KUKA KRL program: MyProgram_205().src

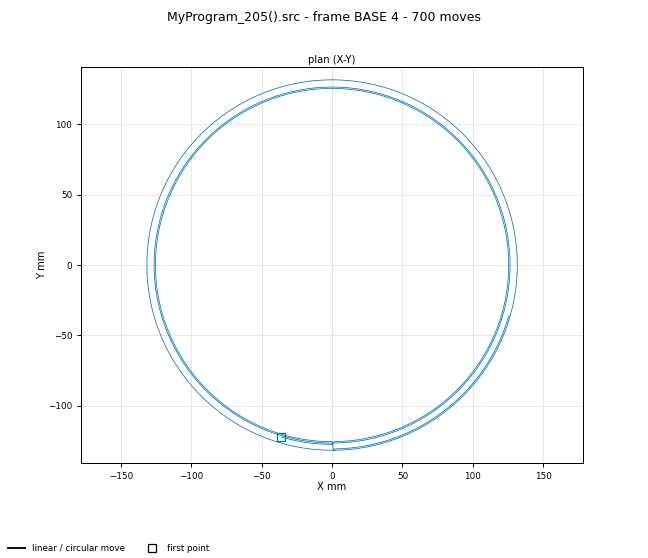
[picture p0: tool path of MyProgram_205().src in frame BASE 4, 700 of 700 moves have a stored position in this frame; points joined in program order, loops and branches not executed]
&ACCESS RVP
&REL 1
&PARAM TEMPLATE = C:\KRC\Roboter\Template\vorgabe
&PARAM EDITMASK = *
DEF MyProgram_205()
; ---- Setting reference (Base) ----
$BASE = BASE_DATA[4]

; --------------------------
; ---- Setting tool (TCP) ----
$TOOL = TOOL_DATA[3]
; --------------------------

$VEL.CP = VEL_APROX_PRINT
Startdeposition()
$VEL.CP = VEL_PRINT
LIN {X -36.0341,Y -122.2263,Z 146,A -108.5004,B 22.4031,C -0.9389,E1 22.3779,E2 195.6452} C_DIS
LIN {X -32.6607,Y -123.1706,Z 146,A -106.9156,B 22.4031,C -0.9383,E1 22.3822,E2 194.0592} C_DIS
LIN {X -28.9305,Y -124.1009,Z 146,A -105.1124,B 22.4031,C -0.9406,E1 22.3871,E2 192.2472} C_DIS
LIN {X -25.3241,Y -124.8856,Z 146,A -103.5291,B 22.4031,C -0.9365,E1 22.3914,E2 190.6725} C_DIS
LIN {X -21.3618,Y -125.6246,Z 146,A -101.0453,B 22.402,C -0.9659,E1 22.3984,E2 188.1089} C_DIS
LIN {X -16.3761,Y -126.3708,Z 146,A -99.4873,B 22.4033,C -0.9336,E1 22.4025,E2 186.6342} C_DIS
LIN {X -12.7363,Y -126.7906,Z 146,A -97.3876,B 22.4025,C -0.9536,E1 22.4085,E2 184.4806} C_DIS
LIN {X -9.0386,Y -127.1067,Z 146,A -96.2108,B 22.4034,C -0.9316,E1 22.4116,E2 183.3613} C_DIS
LIN {X -2.4319,Y -127.4047,Z 146,A -93.38,B 22.4036,C -0.9253,E1 22.4195,E2 180.5461} C_DIS
LIN {X 0.9115,Y -127.3964,Z 146,A -91.8987,B 22.4036,C -0.925,E1 22.4237,E2 179.0657} C_DIS
Enddeposition()
LIN {X 0.9115,Y -127.3964,Z 146,A -91.8987,B 22.4036,C -0.925,E1 22.4237,E2 179.0657} C_DIS
Startdeposition()
$VEL.CP = VEL_PRINT
LIN {X -0.2002,Y -126.4714,Z 146,A -92.567,B 21.3921,C -0.7578,E1 21.404,E2 180.0625} C_DIS
LIN {X -3.5171,Y -126.4217,Z 146,A -94.2559,B 21.3924,C -0.7499,E1 21.3992,E2 181.7734} C_DIS
LIN {X -7.0125,Y -126.2777,Z 146,A -95.5952,B 21.3921,C -0.76,E1 21.3955,E2 183.0853} C_DIS
LIN {X -11.0098,Y -125.9909,Z 146,A -97.3605,B 21.392,C -0.7622,E1 21.3906,E2 184.8454} C_DIS
LIN {X -14.3334,Y -125.6573,Z 146,A -99.0886,B 21.3923,C -0.7535,E1 21.3858,E2 186.5988} C_DIS
LIN {X -19.2644,Y -124.9946,Z 146,A -101.275,B 21.3922,C -0.7568,E1 21.3797,E2 188.778} C_DIS
LIN {X -22.4995,Y -124.4531,Z 146,A -102.727,B 21.3922,C -0.7588,E1 21.3758,E2 190.2264} C_DIS
LIN {X -26.5997,Y -123.6414,Z 146,A -104.6613,B 21.3922,C -0.7579,E1 21.3705,E2 192.1657} C_DIS
LIN {X -29.8792,Y -122.8903,Z 146,A -106.087,B 21.392,C -0.7628,E1 21.3666,E2 193.5803} C_DIS
LIN {X -32.8395,Y -122.1326,Z 146,A -107.6058,B 21.3921,C -0.7581,E1 21.3625,E2 195.1146} C_DIS
LIN {X -37.1654,Y -120.8862,Z 146,A -109.654,B 21.3921,C -0.7592,E1 21.357,E2 197.1639} C_DIS
LIN {X -42.6541,Y -119.0604,Z 146,A -111.9494,B 21.3916,C -0.7746,E1 21.351,E2 199.4219} C_DIS
LIN {X -48.2784,Y -116.8936,Z 146,A -114.7855,B 21.3916,C -0.7729,E1 21.3436,E2 202.27} C_DIS
LIN {X -50.5646,Y -115.9227,Z 146,A -115.9953,B 21.3917,C -0.7707,E1 21.3405,E2 203.4892} C_DIS
LIN {X -53.5348,Y -114.5816,Z 146,A -117.5184,B 21.3917,C -0.7705,E1 21.3366,E2 205.0174} C_DIS
LIN {X -56.4308,Y -113.1836,Z 146,A -118.9521,B 21.3917,C -0.7732,E1 21.333,E2 206.448} C_DIS
LIN {X -59.1321,Y -111.7954,Z 146,A -120.3858,B 21.3917,C -0.7727,E1 21.3294,E2 207.8879} C_DIS
LIN {X -62.7954,Y -109.7812,Z 146,A -122.3752,B 21.3917,C -0.7714,E1 21.3246,E2 209.8876} C_DIS
LIN {X -66.3971,Y -107.6414,Z 146,A -124.2637,B 21.3916,C -0.7746,E1 21.3201,E2 211.7743} C_DIS
LIN {X -69.8004,Y -105.4664,Z 146,A -126.1081,B 21.3915,C -0.7769,E1 21.3157,E2 213.6195} C_DIS
LIN {X -77.0801,Y -100.2691,Z 146,A -129.8585,B 21.3908,C -0.7957,E1 21.3074,E2 217.3336} C_DIS
LIN {X -79.9121,Y -98.0267,Z 146,A -131.4603,B 21.3907,C -0.8001,E1 21.3038,E2 218.9304} C_DIS
LIN {X -83.4451,Y -95.0379,Z 146,A -133.9643,B 21.3911,C -0.788,E1 21.2984,E2 221.4794} C_DIS
LIN {X -86.6555,Y -92.1196,Z 146,A -135.9206,B 21.391,C -0.7923,E1 21.2944,E2 223.4332} C_DIS
LIN {X -89.7097,Y -89.1478,Z 146,A -137.8436,B 21.3908,C -0.7966,E1 21.2906,E2 225.3539} C_DIS
LIN {X -92.795,Y -85.9323,Z 146,A -139.8605,B 21.3906,C -0.8011,E1 21.2867,E2 227.3689} C_DIS
LIN {X -95.6026,Y -82.7974,Z 146,A -141.8312,B 21.3906,C -0.8029,E1 21.2831,E2 229.3453} C_DIS
LIN {X -98.4968,Y -79.3318,Z 146,A -144.1879,B 21.3908,C -0.7956,E1 21.2789,E2 231.7351} C_DIS
LIN {X -100.8297,Y -76.3451,Z 146,A -145.3981,B 21.39,C -0.8194,E1 21.2769,E2 232.8867} C_DIS
LIN {X -103.3227,Y -72.9355,Z 146,A -147.5852,B 21.3902,C -0.8135,E1 21.2733,E2 235.1026} C_DIS
LIN {X -105.7732,Y -69.3344,Z 146,A -149.5373,B 21.39,C -0.8193,E1 21.2703,E2 237.0503} C_DIS
LIN {X -108.0776,Y -65.6847,Z 146,A -151.4874,B 21.3898,C -0.8246,E1 21.2674,E2 238.9977} C_DIS
LIN {X -112.2795,Y -58.2101,Z 146,A -155.097,B 21.389,C -0.8456,E1 21.2626,E2 242.5719} C_DIS
LIN {X -113.9687,Y -54.8262,Z 146,A -156.7959,B 21.3888,C -0.8509,E1 21.2605,E2 244.2672} C_DIS
LIN {X -115.4791,Y -51.568,Z 146,A -158.6195,B 21.3889,C -0.8479,E1 21.2583,E2 246.1109} C_DIS
LIN {X -116.6221,Y -48.9286,Z 146,A -159.9466,B 21.3889,C -0.8507,E1 21.2569,E2 247.4391} C_DIS
LIN {X -117.8749,Y -45.8278,Z 146,A -161.5498,B 21.3888,C -0.8516,E1 21.2552,E2 249.0502} C_DIS
LIN {X -119.1113,Y -42.513,Z 146,A -163.0181,B 21.3884,C -0.8615,E1 21.2538,E2 250.5014} C_DIS
LIN {X -119.9494,Y -40.0857,Z 146,A -164.511,B 21.3888,C -0.8523,E1 21.2525,E2 252.0296} C_DIS
LIN {X -121.4192,Y -35.3851,Z 146,A -166.5476,B 21.3882,C -0.8664,E1 21.2509,E2 254.0414} C_DIS
LIN {X -122.6901,Y -30.6928,Z 146,A -168.844,B 21.3881,C -0.8694,E1 21.2492,E2 256.3453} C_DIS
LIN {X -123.6495,Y -26.5625,Z 146,A -170.6967,B 21.3878,C -0.8779,E1 21.2481,E2 258.1875} C_DIS
LIN {X -124.2918,Y -23.3759,Z 146,A -172.1355,B 21.3875,C -0.8837,E1 21.2473,E2 259.6204} C_DIS
LIN {X -124.9553,Y -19.5185,Z 146,A -173.9521,B 21.3874,C -0.8876,E1 21.2465,E2 261.4393} C_DIS
LIN {X -125.4853,Y -15.7689,Z 146,A -175.8504,B 21.3874,C -0.886,E1 21.2458,E2 263.3554} C_DIS
LIN {X -125.9635,Y -11.3339,Z 146,A -177.6417,B 21.3868,C -0.901,E1 21.2453,E2 265.118} C_DIS
LIN {X -126.1813,Y -8.5712,Z 146,A -179.0869,B 21.387,C -0.8978,E1 21.245,E2 266.5824} C_DIS
LIN {X -126.3845,Y -4.6711,Z 146,A 179.1289,B 21.3868,C -0.9028,E1 21.2448,E2 268.3655} C_DIS
LIN {X -126.4753,Y -0.0344,Z 146,A 177.1063,B 21.3864,C -0.9124,E1 21.2448,E2 270.3762} C_DIS
LIN {X -126.381,Y 4.7613,Z 146,A 174.9068,B 21.3861,C -0.9184,E1 21.2448,E2 272.5751} C_DIS
LIN {X -126.164,Y 8.8087,Z 146,A 173.0434,B 21.3859,C -0.9232,E1 21.2452,E2 274.4385} C_DIS
LIN {X -125.8611,Y 12.4043,Z 146,A 171.377,B 21.3858,C -0.9272,E1 21.2456,E2 276.1058} C_DIS
LIN {X -125.3982,Y 16.4334,Z 146,A 169.5121,B 21.3856,C -0.932,E1 21.2463,E2 277.9708} C_DIS
LIN {X -124.7679,Y 20.6819,Z 146,A 167.6246,B 21.3852,C -0.9403,E1 21.2471,E2 279.8486} C_DIS
LIN {X -124.1633,Y 24.048,Z 146,A 165.628,B 21.3857,C -0.9283,E1 21.2481,E2 281.8923} C_DIS
LIN {X -123.3778,Y 27.7993,Z 146,A 164.5101,B 21.3845,C -0.9571,E1 21.2488,E2 282.9386} C_DIS
LIN {X -122.4488,Y 31.6436,Z 146,A 162.5398,B 21.3845,C -0.9559,E1 21.2501,E2 284.9259} C_DIS
LIN {X -121.5509,Y 34.9355,Z 146,A 160.7569,B 21.3848,C -0.9517,E1 21.2514,E2 286.7326} C_DIS
LIN {X -120.1897,Y 39.3641,Z 146,A 158.9282,B 21.384,C -0.9684,E1 21.253,E2 288.5278} C_DIS
LIN {X -119.2918,Y 42.0064,Z 146,A 157.443,B 21.3842,C -0.9639,E1 21.2543,E2 290.0354} C_DIS
LIN {X -117.8314,Y 45.9397,Z 146,A 155.6344,B 21.3838,C -0.9732,E1 21.2561,E2 291.8306} C_DIS
LIN {X -116.6725,Y 48.808,Z 146,A 153.266,B 21.3852,C -0.941,E1 21.2588,E2 294.3034} C_DIS
LIN {X -114.0463,Y 54.6639,Z 146,A 151.2733,B 21.3834,C -0.9839,E1 21.261,E2 296.1905} C_DIS
LIN {X -111.7773,Y 59.1664,Z 146,A 149.0935,B 21.3829,C -0.9945,E1 21.2638,E2 298.355} C_DIS
LIN {X -110.0652,Y 62.2974,Z 146,A 147.3565,B 21.3829,C -0.9945,E1 21.2662,E2 300.1029} C_DIS
LIN {X -108.057,Y 65.7187,Z 146,A 145.4612,B 21.3829,C -0.9959,E1 21.2689,E2 302.0062} C_DIS
LIN {X -105.7694,Y 69.34,Z 146,A 143.5175,B 21.3826,C -1.0011,E1 21.2718,E2 303.9471} C_DIS
LIN {X -103.2904,Y 72.9812,Z 146,A 141.6623,B 21.3821,C -1.0118,E1 21.2747,E2 305.7835} C_DIS
LIN {X -101.3754,Y 75.6186,Z 146,A 140.0515,B 21.3821,C -1.0106,E1 21.2774,E2 307.407} C_DIS
LIN {X -98.7229,Y 79.051,Z 146,A 138.2823,B 21.3816,C -1.0232,E1 21.2804,E2 309.1514} C_DIS
LIN {X -96.8688,Y 81.3116,Z 146,A 136.7318,B 21.3818,C -1.018,E1 21.2832,E2 310.7249} C_DIS
LIN {X -94.0244,Y 84.5851,Z 146,A 134.6597,B 21.3818,C -1.0187,E1 21.2871,E2 312.806} C_DIS
LIN {X -90.6963,Y 88.1441,Z 146,A 132.5897,B 21.3813,C -1.0293,E1 21.291,E2 314.8575} C_DIS
LIN {X -87.9405,Y 90.8935,Z 146,A 130.7775,B 21.3813,C -1.0316,E1 21.2946,E2 316.6725} C_DIS
LIN {X -85.0052,Y 93.6444,Z 146,A 128.8415,B 21.3813,C -1.0314,E1 21.2986,E2 318.6184} C_DIS
LIN {X -81.8441,Y 96.4194,Z 146,A 127.0047,B 21.3809,C -1.0382,E1 21.3025,E2 320.4449} C_DIS
LIN {X -78.8892,Y 98.8518,Z 146,A 125.3343,B 21.3806,C -1.0443,E1 21.3061,E2 322.1059} C_DIS
LIN {X -75.836,Y 101.2136,Z 146,A 123.5138,B 21.3806,C -1.0451,E1 21.3101,E2 323.932} C_DIS
LIN {X -71.8456,Y 104.084,Z 146,A 121.2314,B 21.3805,C -1.0473,E1 21.3154,E2 326.2177} C_DIS
LIN {X -68.6655,Y 106.2086,Z 146,A 119.5061,B 21.3803,C -1.0509,E1 21.3194,E2 327.94} C_DIS
LIN {X -65.3364,Y 108.2881,Z 146,A 117.7441,B 21.3801,C -1.0547,E1 21.3236,E2 329.698} C_DIS
LIN {X -62.0308,Y 110.215,Z 146,A 116.0512,B 21.3799,C -1.0593,E1 21.3277,E2 331.3842} C_DIS
LIN {X -58.7576,Y 111.992,Z 146,A 114.4151,B 21.3797,C -1.0641,E1 21.3317,E2 333.0126} C_DIS
LIN {X -55.9636,Y 113.414,Z 146,A 112.9155,B 21.3797,C -1.0632,E1 21.3354,E2 334.5194} C_DIS
LIN {X -52.2563,Y 115.1712,Z 146,A 111.1648,B 21.3794,C -1.0702,E1 21.3398,E2 336.256} C_DIS
LIN {X -49.3423,Y 116.4493,Z 146,A 109.7278,B 21.3794,C -1.0724,E1 21.3435,E2 337.691} C_DIS
LIN {X -46.2318,Y 117.7179,Z 146,A 107.792,B 21.38,C -1.0581,E1 21.3486,E2 339.6712} C_DIS
LIN {X -43.1661,Y 118.8758,Z 146,A 106.861,B 21.3789,C -1.0818,E1 21.3509,E2 340.5391} C_DIS
LIN {X -38.6181,Y 120.4299,Z 146,A 104.0568,B 21.3799,C -1.0595,E1 21.3585,E2 343.4109} C_DIS
LIN {X -35.1143,Y 121.4985,Z 146,A 102.8457,B 21.379,C -1.079,E1 21.3616,E2 344.5707} C_DIS
LIN {X -32.1662,Y 122.3121,Z 146,A 101.4603,B 21.379,C -1.0804,E1 21.3654,E2 345.9548} C_DIS
LIN {X -29.4254,Y 122.9997,Z 146,A 100.0934,B 21.379,C -1.0781,E1 21.3691,E2 347.3303} C_DIS
LIN {X -26.4415,Y 123.6756,Z 146,A 98.758,B 21.3789,C -1.0813,E1 21.3727,E2 348.6589} C_DIS
LIN {X -23.5848,Y 124.2519,Z 146,A 97.3859,B 21.3789,C -1.0802,E1 21.3765,E2 350.0358} C_DIS
LIN {X -19.2825,Y 124.9918,Z 146,A 95.384,B 21.3789,C -1.0806,E1 21.382,E2 352.0388} C_DIS
LIN {X -14.8809,Y 125.592,Z 146,A 93.3443,B 21.3789,C -1.0806,E1 21.3877,E2 354.0802} C_DIS
LIN {X -11.5392,Y 125.9442,Z 146,A 91.8914,B 21.3787,C -1.0841,E1 21.3917,E2 355.5245} C_DIS
LIN {X -7.5118,Y 126.2475,Z 146,A 90.1618,B 21.3785,C -1.0889,E1 21.3965,E2 357.2417} C_DIS
LIN {X -4.6049,Y 126.3871,Z 146,A 88.8159,B 21.3785,C -1.0882,E1 21.4002,E2 358.5899} C_DIS
LIN {X -1.3758,Y 126.4649,Z 146,A 87.2194,B 21.3788,C -1.083,E1 21.4047,E2 360.2007} C_DIS
LIN {X 2.7721,Y 126.4415,Z 146,A 85.4789,B 21.3785,C -1.0889,E1 21.4095,E2 361.9247} C_DIS
LIN {X 7.4851,Y 126.2492,Z 146,A 83.1677,B 21.3789,C -1.0818,E1 21.416,E2 364.2545} C_DIS
LIN {X 11.0113,Y 125.9908,Z 146,A 81.7032,B 21.3786,C -1.0873,E1 21.4201,E2 365.703} C_DIS
LIN {X 14.5679,Y 125.6293,Z 146,A 79.9193,B 21.3789,C -1.0802,E1 21.4251,E2 367.5049} C_DIS
LIN {X 18.102,Y 125.1684,Z 146,A 78.4196,B 21.3787,C -1.0845,E1 21.4292,E2 368.9912} C_DIS
LIN {X 22.1034,Y 124.524,Z 146,A 76.484,B 21.379,C -1.0798,E1 21.4345,E2 370.9376} C_DIS
LIN {X 25.5845,Y 123.856,Z 146,A 75.0215,B 21.3787,C -1.085,E1 21.4385,E2 372.3837} C_DIS
LIN {X 28.2648,Y 123.2714,Z 146,A 73.7554,B 21.3787,C -1.0833,E1 21.4419,E2 373.6523} C_DIS
LIN {X 31.3296,Y 122.5285,Z 146,A 72.3059,B 21.3789,C -1.0816,E1 21.4459,E2 375.1039} C_DIS
LIN {X 35.1324,Y 121.4932,Z 146,A 70.4772,B 21.379,C -1.0785,E1 21.4508,E2 376.9375} C_DIS
LIN {X 39.9482,Y 119.9952,Z 146,A 68.5858,B 21.3783,C -1.0932,E1 21.4557,E2 378.7844} C_DIS
LIN {X 45.5483,Y 117.9836,Z 146,A 65.7798,B 21.3787,C -1.0861,E1 21.4632,E2 381.6031} C_DIS
LIN {X 48.8944,Y 116.6364,Z 146,A 63.9332,B 21.3792,C -1.0754,E1 21.468,E2 383.474} C_DIS
LIN {X 52.184,Y 115.2036,Z 146,A 62.3271,B 21.3792,C -1.0743,E1 21.4721,E2 385.0783} C_DIS
LIN {X 54.7767,Y 113.9924,Z 146,A 61.0283,B 21.3792,C -1.0727,E1 21.4753,E2 386.3776} C_DIS
LIN {X 58.1819,Y 112.2943,Z 146,A 59.1911,B 21.3796,C -1.0656,E1 21.48,E2 388.2281} C_DIS
LIN {X 62.1945,Y 110.123,Z 146,A 57.2128,B 21.3796,C -1.0665,E1 21.4848,E2 390.1971} C_DIS
LIN {X 65.5406,Y 108.1647,Z 146,A 55.509,B 21.3796,C -1.0661,E1 21.4888,E2 391.8956} C_DIS
LIN {X 68.6592,Y 106.2127,Z 146,A 53.774,B 21.3799,C -1.0606,E1 21.493,E2 393.639} C_DIS
LIN {X 71.951,Y 104.0112,Z 146,A 51.9083,B 21.3802,C -1.0546,E1 21.4973,E2 395.5138} C_DIS
LIN {X 75.3343,Y 101.5872,Z 146,A 50.0448,B 21.3802,C -1.0522,E1 21.5015,E2 397.3757} C_DIS
LIN {X 78.1149,Y 99.4646,Z 146,A 48.5612,B 21.3802,C -1.0537,E1 21.5047,E2 398.8488} C_DIS
LIN {X 80.9804,Y 97.1467,Z 146,A 46.7924,B 21.3805,C -1.0463,E1 21.5086,E2 400.6299} C_DIS
LIN {X 84.3041,Y 94.2761,Z 146,A 44.8386,B 21.3807,C -1.0439,E1 21.5127,E2 402.581} C_DIS
LIN {X 87.2293,Y 91.5764,Z 146,A 43.0399,B 21.3808,C -1.0404,E1 21.5163,E2 404.3804} C_DIS
LIN {X 90.1747,Y 88.6775,Z 146,A 41.2654,B 21.3808,C -1.0407,E1 21.5198,E2 406.1452} C_DIS
LIN {X 92.9177,Y 85.7994,Z 146,A 39.5495,B 21.3808,C -1.0404,E1 21.5231,E2 407.853} C_DIS
LIN {X 95.3156,Y 83.127,Z 146,A 37.7882,B 21.3813,C -1.0309,E1 21.5264,E2 409.6309} C_DIS
LIN {X 98.1919,Y 79.7099,Z 146,A 35.7281,B 21.3815,C -1.0245,E1 21.5301,E2 411.697} C_DIS
LIN {X 100.9079,Y 76.2415,Z 146,A 33.8091,B 21.3816,C -1.0231,E1 21.5333,E2 413.6092} C_DIS
LIN {X 103.467,Y 72.7309,Z 146,A 31.953,B 21.3816,C -1.0231,E1 21.5363,E2 415.4545} C_DIS
LIN {X 105.205,Y 70.193,Z 146,A 30.5018,B 21.3819,C -1.0171,E1 21.5386,E2 416.9137} C_DIS
LIN {X 107.5118,Y 66.6065,Z 146,A 28.6131,B 21.382,C -1.0139,E1 21.5414,E2 418.7996} C_DIS
LIN {X 109.4763,Y 63.3254,Z 146,A 26.7412,B 21.3825,C -1.0032,E1 21.5441,E2 420.6892} C_DIS
LIN {X 111.3301,Y 60.0067,Z 146,A 25.0158,B 21.3827,C -0.9984,E1 21.5464,E2 422.417} C_DIS
LIN {X 113.4712,Y 55.8477,Z 146,A 23.0715,B 21.3827,C -1.0003,E1 21.5488,E2 424.3438} C_DIS
LIN {X 114.9056,Y 52.8341,Z 146,A 21.6136,B 21.3827,C -0.9985,E1 21.5506,E2 425.7974} C_DIS
LIN {X 117.6429,Y 46.4246,Z 146,A 18.5231,B 21.383,C -0.9924,E1 21.5539,E2 428.8843} C_DIS
LIN {X 118.6502,Y 43.7857,Z 146,A 17.204,B 21.3832,C -0.9869,E1 21.5552,E2 430.2096} C_DIS
LIN {X 119.597,Y 41.1262,Z 146,A 15.6046,B 21.384,C -0.9689,E1 21.5567,E2 431.8474} C_DIS
LIN {X 121.2732,Y 35.884,Z 146,A 13.3951,B 21.3838,C -0.9741,E1 21.5585,E2 434.0279} C_DIS
LIN {X 122.1777,Y 32.6703,Z 146,A 11.93,B 21.3839,C -0.9716,E1 21.5596,E2 435.4896} C_DIS
LIN {X 122.9913,Y 29.4602,Z 146,A 10.424,B 21.3841,C -0.9668,E1 21.5606,E2 436.9984} C_DIS
LIN {X 123.696,Y 26.347,Z 146,A 9.0665,B 21.3841,C -0.9663,E1 21.5614,E2 438.3478} C_DIS
LIN {X 124.2447,Y 23.6226,Z 146,A 7.7618,B 21.3844,C -0.9604,E1 21.5621,E2 439.6596} C_DIS
LIN {X 124.8827,Y 19.9873,Z 146,A 6.1731,B 21.3844,C -0.9589,E1 21.5628,E2 441.2413} C_DIS
LIN {X 125.3847,Y 16.5368,Z 146,A 4.5913,B 21.3847,C -0.9539,E1 21.5635,E2 442.8256} C_DIS
LIN {X 125.8017,Y 13,Z 146,A 2.9894,B 21.3849,C -0.9494,E1 21.564,E2 444.4287} C_DIS
LIN {X 126.0952,Y 9.751,Z 146,A 1.5779,B 21.3849,C -0.9477,E1 21.5643,E2 445.8348} C_DIS
LIN {X 126.2638,Y 7.2469,Z 146,A 0.1224,B 21.3857,C -0.9298,E1 21.5645,E2 447.3287} C_DIS
LIN {X 126.4447,Y 2.6084,Z 146,A -1.8242,B 21.3857,C -0.9301,E1 21.5647,E2 449.2606} C_DIS
LIN {X 126.4634,Y -1.4399,Z 146,A -3.6754,B 21.3859,C -0.9235,E1 21.5647,E2 451.1168} C_DIS
LIN {X 126.3687,Y -5.0768,Z 146,A -5.2969,B 21.3861,C -0.9195,E1 21.5645,E2 452.7378} C_DIS
LIN {X 126.1804,Y -8.5843,Z 146,A -6.8164,B 21.3861,C -0.9176,E1 21.5643,E2 454.2516} C_DIS
LIN {X 125.9003,Y -11.996,Z 146,A -8.3839,B 21.3864,C -0.912,E1 21.5639,E2 455.8235} C_DIS
LIN {X 125.3751,Y -16.6097,Z 146,A -10.2401,B 21.3862,C -0.9164,E1 21.5633,E2 457.6546} C_DIS
LIN {X 124.9979,Y -19.2433,Z 146,A -11.6731,B 21.3868,C -0.9023,E1 21.5627,E2 459.1159} C_DIS
LIN {X 124.3558,Y -23.0412,Z 146,A -13.296,B 21.3868,C -0.9023,E1 21.5619,E2 460.7276} C_DIS
LIN {X 123.5962,Y -26.8094,Z 146,A -15.1438,B 21.3872,C -0.892,E1 21.5608,E2 462.5906} C_DIS
LIN {X 122.793,Y -30.2827,Z 146,A -16.6457,B 21.3872,C -0.892,E1 21.5599,E2 464.0822} C_DIS
LIN {X 121.8501,Y -33.8719,Z 146,A -18.8983,B 21.3884,C -0.8613,E1 21.5582,E2 466.4032} C_DIS
LIN {X 120.5843,Y -38.135,Z 146,A -20.1527,B 21.3873,C -0.889,E1 21.5572,E2 467.5734} C_DIS
LIN {X 119.7154,Y -40.7847,Z 146,A -21.5355,B 21.3877,C -0.8797,E1 21.556,E2 468.9723} C_DIS
LIN {X 118.3362,Y -44.6241,Z 146,A -23.4349,B 21.388,C -0.8718,E1 21.5541,E2 470.8806} C_DIS
LIN {X 116.8715,Y -48.3314,Z 146,A -25.6354,B 21.3889,C -0.8487,E1 21.5518,E2 473.1295} C_DIS
LIN {X 115.422,Y -51.6956,Z 146,A -26.9406,B 21.3885,C -0.8596,E1 21.5503,E2 474.3967} C_DIS
LIN {X 113.7971,Y -55.1856,Z 146,A -28.5736,B 21.3885,C -0.8594,E1 21.5484,E2 476.0198} C_DIS
LIN {X 112.5392,Y -57.7039,Z 146,A -29.9715,B 21.3888,C -0.8502,E1 21.5466,E2 477.4339} C_DIS
LIN {X 110.82,Y -60.9443,Z 146,A -31.6223,B 21.389,C -0.8459,E1 21.5444,E2 479.0863} C_DIS
LIN {X 109.0869,Y -63.9939,Z 146,A -33.1803,B 21.3891,C -0.8427,E1 21.5422,E2 480.6432} C_DIS
LIN {X 106.8228,Y -67.7059,Z 146,A -35.435,B 21.3898,C -0.8246,E1 21.5388,E2 482.9339} C_DIS
LIN {X 104.8688,Y -70.6948,Z 146,A -36.6955,B 21.3894,C -0.836,E1 21.5369,E2 484.1559} C_DIS
LIN {X 103.3679,Y -72.8713,Z 146,A -37.9082,B 21.3895,C -0.832,E1 21.535,E2 485.3722} C_DIS
LIN {X 100.9849,Y -76.1393,Z 146,A -39.9844,B 21.3901,C -0.8163,E1 21.5315,E2 487.4794} C_DIS
LIN {X 99.006,Y -78.6955,Z 146,A -41.1237,B 21.3897,C -0.8269,E1 21.5296,E2 488.5834} C_DIS
LIN {X 94.5241,Y -84.0266,Z 146,A -44.3113,B 21.39,C -0.8174,E1 21.5238,E2 491.7797} C_DIS
LIN {X 89.5198,Y -89.3389,Z 146,A -48.2395,B 21.3913,C -0.7821,E1 21.516,E2 495.7843} C_DIS
LIN {X 85.8463,Y -92.8744,Z 146,A -49.9498,B 21.3906,C -0.803,E1 21.5127,E2 497.4291} C_DIS
LIN {X 80.2118,Y -97.7817,Z 146,A -53.6721,B 21.3914,C -0.7807,E1 21.5046,E2 501.1951} C_DIS
LIN {X 77.1053,Y -100.2499,Z 146,A -55.1228,B 21.391,C -0.7921,E1 21.5015,E2 502.6084} C_DIS
LIN {X 72.465,Y -103.6536,Z 146,A -57.5038,B 21.3908,C -0.7967,E1 21.4962,E2 504.9667} C_DIS
LIN {X 70.5141,Y -104.9907,Z 146,A -58.7664,B 21.3912,C -0.7863,E1 21.4932,E2 506.2528} C_DIS
LIN {X 66.9866,Y -107.2753,Z 146,A -60.6679,B 21.3912,C -0.7828,E1 21.4887,E2 508.1564} C_DIS
LIN {X 63.1023,Y -109.6054,Z 146,A -62.7171,B 21.3914,C -0.7793,E1 21.4838,E2 510.2079} C_DIS
LIN {X 59.0055,Y -111.8619,Z 146,A -64.5512,B 21.3911,C -0.7881,E1 21.4794,E2 512.0115} C_DIS
LIN {X 56.6188,Y -113.0908,Z 146,A -66.0383,B 21.3916,C -0.7743,E1 21.4756,E2 513.5314} C_DIS
LIN {X 50.8017,Y -115.8202,Z 146,A -69.0261,B 21.3918,C -0.7666,E1 21.468,E2 516.5313} C_DIS
LIN {X 46.9994,Y -117.4131,Z 146,A -70.7002,B 21.3916,C -0.7724,E1 21.4637,E2 518.185} C_DIS
LIN {X 43.1653,Y -118.8761,Z 146,A -73.0884,B 21.3925,C -0.7473,E1 21.4573,E2 520.6359} C_DIS
LIN {X 38.9648,Y -120.3192,Z 146,A -74.4068,B 21.3916,C -0.7746,E1 21.454,E2 521.8766} C_DIS
LIN {X 35.1139,Y -121.4987,Z 146,A -76.4604,B 21.392,C -0.7628,E1 21.4484,E2 523.9584} C_DIS
LIN {X 31.224,Y -122.5553,Z 146,A -78.2182,B 21.392,C -0.7639,E1 21.4437,E2 525.7099} C_DIS
LIN {X 27.7361,Y -123.3922,Z 146,A -79.9259,B 21.3921,C -0.7588,E1 21.439,E2 527.4285} C_DIS
LIN {X 23.6769,Y -124.2343,Z 146,A -81.6893,B 21.392,C -0.7622,E1 21.4342,E2 529.1802} C_DIS
LIN {X 20.477,Y -124.8021,Z 146,A -83.2544,B 21.3922,C -0.7572,E1 21.4299,E2 530.757} C_DIS
LIN {X 16.4443,Y -125.3968,Z 146,A -84.764,B 21.3917,C -0.7703,E1 21.4258,E2 532.2292} C_DIS
LIN {X 13.6399,Y -125.7328,Z 146,A -86.2982,B 21.3921,C -0.7587,E1 21.4215,E2 533.7936} C_DIS
LIN {X 9.6443,Y -126.103,Z 146,A -88.2666,B 21.3924,C -0.7515,E1 21.4159,E2 535.7805} C_DIS
LIN {X 3.5217,Y -126.4215,Z 146,A -90.838,B 21.3921,C -0.7593,E1 21.4088,E2 538.3297} C_DIS
LIN {X 0.9047,Y -126.4634,Z 146,A -91.6983,B 21.3916,C -0.7727,E1 21.4065,E2 539.153} C_DIS
Enddeposition()
LIN {X 0.9047,Y -126.4634,Z 146,A -91.6983,B 21.3916,C -0.7727,E1 21.4065,E2 539.153} C_DIS
Startdeposition()
$VEL.CP = VEL_PRINT
LIN {X 1.5275,Y -125.5056,Z 146,A -90.6951,B 20.265,C -0.6363,E1 20.2782,E2 538.4061} C_DIS
LIN {X 4.5983,Y -125.4297,Z 146,A -89.3182,B 20.265,C -0.6358,E1 20.282,E2 537.0313} C_DIS
LIN {X 7.9101,Y -125.2642,Z 146,A -87.8871,B 20.265,C -0.633,E1 20.286,E2 535.6088} C_DIS
LIN {X 11.0165,Y -125.03,Z 146,A -86.458,B 20.265,C -0.6339,E1 20.29,E2 534.178} C_DIS
LIN {X 13.8261,Y -124.7503,Z 146,A -85.1681,B 20.265,C -0.6347,E1 20.2936,E2 532.8871} C_DIS
LIN {X 17.1185,Y -124.3423,Z 146,A -83.6966,B 20.265,C -0.6338,E1 20.2976,E2 531.4196} C_DIS
LIN {X 19.9422,Y -123.9212,Z 146,A -82.2521,B 20.2649,C -0.6404,E1 20.3016,E2 529.9579} C_DIS
LIN {X 22.9726,Y -123.3947,Z 146,A -80.86,B 20.2649,C -0.641,E1 20.3055,E2 528.566} C_DIS
LIN {X 26.2347,Y -122.7413,Z 146,A -79.4247,B 20.2649,C -0.6389,E1 20.3094,E2 527.1391} C_DIS
LIN {X 29.2363,Y -122.0609,Z 146,A -77.8981,B 20.2647,C -0.6451,E1 20.3136,E2 525.5972} C_DIS
LIN {X 33.477,Y -120.9669,Z 146,A -75.967,B 20.2647,C -0.6443,E1 20.3188,E2 523.6723} C_DIS
LIN {X 36.6722,Y -120.0364,Z 146,A -74.4493,B 20.2647,C -0.6459,E1 20.3228,E2 522.1534} C_DIS
LIN {X 40.6153,Y -118.7613,Z 146,A -72.5021,B 20.2645,C -0.6504,E1 20.328,E2 520.198} C_DIS
LIN {X 44.6291,Y -117.3125,Z 146,A -70.5422,B 20.2645,C -0.6534,E1 20.3331,E2 518.2349} C_DIS
LIN {X 48.0208,Y -115.9642,Z 146,A -69.0325,B 20.2645,C -0.6492,E1 20.337,E2 516.7414} C_DIS
LIN {X 50.8395,Y -114.7567,Z 146,A -67.6403,B 20.2645,C -0.6509,E1 20.3406,E2 515.3486} C_DIS
LIN {X 53.6272,Y -113.481,Z 146,A -66.1493,B 20.2644,C -0.6568,E1 20.3444,E2 513.8455} C_DIS
LIN {X 56.4311,Y -112.1133,Z 146,A -64.7483,B 20.2644,C -0.6581,E1 20.3479,E2 512.4456} C_DIS
LIN {X 59.1794,Y -110.6882,Z 146,A -63.4186,B 20.2644,C -0.6569,E1 20.3511,E2 511.124} C_DIS
LIN {X 62.0908,Y -109.0815,Z 146,A -61.9056,B 20.2643,C -0.6593,E1 20.3548,E2 509.6097} C_DIS
LIN {X 64.743,Y -107.5287,Z 146,A -60.5114,B 20.2643,C -0.6614,E1 20.3582,E2 508.2149} C_DIS
LIN {X 67.356,Y -105.9119,Z 146,A -59.1411,B 20.2642,C -0.6626,E1 20.3614,E2 506.8466} C_DIS
LIN {X 69.7222,Y -104.3688,Z 146,A -57.8273,B 20.2641,C -0.6661,E1 20.3645,E2 505.5284} C_DIS
LIN {X 72.4607,Y -102.4865,Z 146,A -56.3443,B 20.2641,C -0.6676,E1 20.3679,E2 504.0474} C_DIS
LIN {X 75.1801,Y -100.5089,Z 146,A -54.7136,B 20.2638,C -0.6747,E1 20.3716,E2 502.4036} C_DIS
LIN {X 78.407,Y -98.0125,Z 146,A -52.7786,B 20.2636,C -0.6817,E1 20.3758,E2 500.4577} C_DIS
LIN {X 81.9309,Y -95.086,Z 146,A -50.838,B 20.2636,C -0.6799,E1 20.3799,E2 498.5316} C_DIS
LIN {X 84.8351,Y -92.5042,Z 146,A -48.9821,B 20.2634,C -0.6874,E1 20.3838,E2 496.6638} C_DIS
LIN {X 87.9069,Y -89.5901,Z 146,A -47.1348,B 20.2634,C -0.6882,E1 20.3875,E2 494.8237} C_DIS
LIN {X 90.5654,Y -86.9022,Z 146,A -45.3266,B 20.2631,C -0.6958,E1 20.3911,E2 493.0035} C_DIS
LIN {X 93.5066,Y -83.7289,Z 146,A -43.3575,B 20.263,C -0.7004,E1 20.3948,E2 491.0321} C_DIS
LIN {X 96.4415,Y -80.3317,Z 146,A -41.4313,B 20.263,C -0.7004,E1 20.3982,E2 489.1173} C_DIS
LIN {X 98.5642,Y -77.7121,Z 146,A -39.8065,B 20.2627,C -0.708,E1 20.4011,E2 487.4802} C_DIS
LIN {X 100.9647,Y -74.567,Z 146,A -38.0791,B 20.2627,C -0.7094,E1 20.404,E2 485.7592} C_DIS
LIN {X 102.7543,Y -72.081,Z 146,A -36.7434,B 20.2627,C -0.7104,E1 20.4061,E2 484.4286} C_DIS
LIN {X 104.4818,Y -69.5529,Z 146,A -35.4112,B 20.2626,C -0.7115,E1 20.4082,E2 483.1018} C_DIS
LIN {X 106.0149,Y -67.1932,Z 146,A -34.0091,B 20.2623,C -0.72,E1 20.4103,E2 481.6842} C_DIS
LIN {X 107.6582,Y -64.5278,Z 146,A -32.6711,B 20.2623,C -0.72,E1 20.4122,E2 480.3545} C_DIS
LIN {X 109.3293,Y -61.6535,Z 146,A -31.1623,B 20.2622,C -0.724,E1 20.4143,E2 478.8443} C_DIS
LIN {X 110.6892,Y -59.1777,Z 146,A -29.8206,B 20.262,C -0.7299,E1 20.4161,E2 477.4945} C_DIS
LIN {X 112.3937,Y -55.8689,Z 146,A -28.35,B 20.2621,C -0.7251,E1 20.418,E2 476.0476} C_DIS
LIN {X 113.5721,Y -53.4366,Z 146,A -26.9607,B 20.2618,C -0.7353,E1 20.4197,E2 474.6385} C_DIS
LIN {X 115.0827,Y -50.0962,Z 146,A -25.4929,B 20.2619,C -0.7314,E1 20.4213,E2 473.1918} C_DIS
LIN {X 116.0604,Y -47.7905,Z 146,A -24.1797,B 20.2615,C -0.7421,E1 20.4228,E2 471.8571} C_DIS
LIN {X 117.3154,Y -44.6213,Z 146,A -22.4509,B 20.2611,C -0.7541,E1 20.4245,E2 470.1059} C_DIS
LIN {X 118.7635,Y -40.6089,Z 146,A -20.6948,B 20.2611,C -0.7519,E1 20.4261,E2 468.3687} C_DIS
LIN {X 119.6497,Y -37.916,Z 146,A -19.4151,B 20.2611,C -0.7552,E1 20.4272,E2 467.0886} C_DIS
LIN {X 120.5977,Y -34.7855,Z 146,A -17.7717,B 20.2607,C -0.7662,E1 20.4285,E2 465.4255} C_DIS
LIN {X 121.6577,Y -30.8705,Z 146,A -16.0336,B 20.2607,C -0.7671,E1 20.4298,E2 463.6976} C_DIS
LIN {X 122.4658,Y -27.4945,Z 146,A -14.5273,B 20.2606,C -0.7686,E1 20.4307,E2 462.1978} C_DIS
LIN {X 123.1529,Y -24.2374,Z 146,A -13.05,B 20.2605,C -0.7715,E1 20.4315,E2 460.723} C_DIS
LIN {X 123.7096,Y -21.21,Z 146,A -11.6125,B 20.2603,C -0.7773,E1 20.4322,E2 459.2795} C_DIS
LIN {X 124.156,Y -18.4221,Z 146,A -10.253,B 20.26,C -0.7844,E1 20.4328,E2 457.9099} C_DIS
LIN {X 124.6014,Y -15.1062,Z 146,A -8.8954,B 20.26,C -0.7819,E1 20.4333,E2 456.5693} C_DIS
LIN {X 124.9098,Y -12.3001,Z 146,A -7.4878,B 20.2598,C -0.7911,E1 20.4337,E2 455.1461} C_DIS
LIN {X 125.1733,Y -9.2358,Z 146,A -6.1556,B 20.2598,C -0.7924,E1 20.434,E2 453.82} C_DIS
LIN {X 125.3746,Y -5.918,Z 146,A -4.6899,B 20.2596,C -0.795,E1 20.4342,E2 452.3579} C_DIS
LIN {X 125.4838,Y -2.8162,Z 146,A -3.2269,B 20.2594,C -0.8014,E1 20.4343,E2 450.8874} C_DIS
LIN {X 125.5153,Y 0.4415,Z 146,A -1.5839,B 20.2589,C -0.8128,E1 20.4343,E2 449.2242} C_DIS
LIN {X 125.4292,Y 4.6123,Z 146,A 0.1801,B 20.2589,C -0.8128,E1 20.4342,E2 447.4735} C_DIS
LIN {X 125.262,Y 7.9468,Z 146,A 1.5871,B 20.2589,C -0.8125,E1 20.434,E2 446.0777} C_DIS
LIN {X 125.0293,Y 11.0249,Z 146,A 3.015,B 20.2587,C -0.8177,E1 20.4336,E2 444.6456} C_DIS
LIN {X 124.7494,Y 13.8348,Z 146,A 4.4518,B 20.2583,C -0.828,E1 20.4332,E2 443.1899} C_DIS
LIN {X 124.34,Y 17.1345,Z 146,A 5.7555,B 20.2585,C -0.8236,E1 20.4327,E2 441.9088} C_DIS
LIN {X 123.9235,Y 19.9279,Z 146,A 7.2531,B 20.258,C -0.8364,E1 20.4321,E2 440.3853} C_DIS
LIN {X 123.3937,Y 22.9776,Z 146,A 8.5763,B 20.258,C -0.8369,E1 20.4314,E2 439.0705} C_DIS
LIN {X 122.74,Y 26.2404,Z 146,A 10.004,B 20.258,C -0.8377,E1 20.4306,E2 437.6511} C_DIS
LIN {X 121.9093,Y 29.8652,Z 146,A 11.8275,B 20.2575,C -0.8482,E1 20.4294,E2 435.8109} C_DIS
LIN {X 120.9664,Y 33.4788,Z 146,A 13.4415,B 20.2575,C -0.8494,E1 20.4282,E2 434.205} C_DIS
LIN {X 119.9256,Y 37.034,Z 146,A 15.1782,B 20.2572,C -0.8564,E1 20.4268,E2 432.4609} C_DIS
LIN {X 118.6018,Y 41.0755,Z 146,A 16.9816,B 20.2572,C -0.8562,E1 20.4252,E2 430.6708} C_DIS
LIN {X 117.4892,Y 44.1574,Z 146,A 18.4261,B 20.2572,C -0.8583,E1 20.4239,E2 429.2303} C_DIS
LIN {X 116.5453,Y 46.5926,Z 146,A 19.647,B 20.2569,C -0.863,E1 20.4226,E2 428.0047} C_DIS
LIN {X 115.3723,Y 49.4262,Z 146,A 21.047,B 20.2568,C -0.8669,E1 20.4211,E2 426.603} C_DIS
LIN {X 114.1128,Y 52.2688,Z 146,A 22.4454,B 20.2567,C -0.87,E1 20.4195,E2 425.2053} C_DIS
LIN {X 112.7974,Y 55.0506,Z 146,A 23.8377,B 20.2565,C -0.8734,E1 20.4178,E2 423.8129} C_DIS
LIN {X 111.2118,Y 58.1851,Z 146,A 25.4518,B 20.2563,C -0.8782,E1 20.4157,E2 422.1957} C_DIS
LIN {X 109.2045,Y 61.8752,Z 146,A 27.4028,B 20.256,C -0.8847,E1 20.4131,E2 420.2389} C_DIS
LIN {X 107.3785,Y 64.9913,Z 146,A 28.9029,B 20.2561,C -0.8828,E1 20.411,E2 418.754} C_DIS
LIN {X 105.5619,Y 67.9026,Z 146,A 30.6734,B 20.2556,C -0.8954,E1 20.4083,E2 416.9586} C_DIS
LIN {X 103.4986,Y 71.0074,Z 146,A 32.2734,B 20.2556,C -0.8954,E1 20.4058,E2 415.3686} C_DIS
LIN {X 101.7285,Y 73.5211,Z 146,A 33.6738,B 20.2555,C -0.8987,E1 20.4035,E2 413.9672} C_DIS
LIN {X 99.341,Y 76.7165,Z 146,A 35.5541,B 20.2552,C -0.9056,E1 20.4003,E2 412.0785} C_DIS
LIN {X 96.5353,Y 80.2184,Z 146,A 37.5768,B 20.255,C -0.9093,E1 20.3968,E2 410.057} C_DIS
LIN {X 93.9447,Y 83.2372,Z 146,A 39.4026,B 20.2548,C -0.9138,E1 20.3934,E2 408.2286} C_DIS
LIN {X 90.9858,Y 86.4623,Z 146,A 41.4158,B 20.2546,C -0.9188,E1 20.3895,E2 406.2121} C_DIS
LIN {X 88.1176,Y 89.3835,Z 146,A 43.2705,B 20.2544,C -0.9221,E1 20.3859,E2 404.3576} C_DIS
LIN {X 84.7744,Y 92.5601,Z 146,A 45.348,B 20.2544,C -0.9253,E1 20.3816,E2 402.2819} C_DIS
LIN {X 81.606,Y 95.3658,Z 146,A 47.2334,B 20.2542,C -0.9271,E1 20.3777,E2 400.4006} C_DIS
LIN {X 78.4298,Y 97.9944,Z 146,A 49.1616,B 20.254,C -0.9325,E1 20.3735,E2 398.466} C_DIS
LIN {X 74.7759,Y 100.8098,Z 146,A 51.1086,B 20.2541,C -0.9297,E1 20.3692,E2 396.536} C_DIS
LIN {X 72.0588,Y 102.77,Z 146,A 52.6302,B 20.2541,C -0.932,E1 20.3657,E2 395.0145} C_DIS
LIN {X 69.5193,Y 104.5041,Z 146,A 53.9734,B 20.2541,C -0.9318,E1 20.3626,E2 393.6776} C_DIS
LIN {X 66.8157,Y 106.2531,Z 146,A 55.4026,B 20.254,C -0.9325,E1 20.3593,E2 392.2524} C_DIS
LIN {X 63.9036,Y 108.0301,Z 146,A 57.2038,B 20.2534,C -0.9447,E1 20.3549,E2 390.423} C_DIS
LIN {X 60.3039,Y 110.0796,Z 146,A 59.0263,B 20.2534,C -0.9446,E1 20.3505,E2 388.6077} C_DIS
LIN {X 57.5731,Y 111.5319,Z 146,A 60.3207,B 20.2536,C -0.9417,E1 20.3473,E2 387.3262} C_DIS
LIN {X 54.8229,Y 112.9097,Z 146,A 61.7365,B 20.2535,C -0.9439,E1 20.3438,E2 385.9088} C_DIS
LIN {X 52.0374,Y 114.2198,Z 146,A 63.2901,B 20.2531,C -0.9515,E1 20.3398,E2 384.3381} C_DIS
LIN {X 49.225,Y 115.4593,Z 146,A 64.5325,B 20.2534,C -0.9466,E1 20.3366,E2 383.1137} C_DIS
LIN {X 46.6111,Y 116.5379,Z 146,A 65.8169,B 20.2534,C -0.9477,E1 20.3333,E2 381.8298} C_DIS
LIN {X 43.7234,Y 117.6517,Z 146,A 67.2251,B 20.2533,C -0.9489,E1 20.3296,E2 380.422} C_DIS
LIN {X 40.5981,Y 118.7672,Z 146,A 68.736,B 20.2533,C -0.9501,E1 20.3256,E2 378.9116} C_DIS
LIN {X 37.7582,Y 119.7,Z 146,A 70.2582,B 20.2529,C -0.9575,E1 20.3216,E2 377.3716} C_DIS
LIN {X 34.7176,Y 120.6176,Z 146,A 71.5422,B 20.2531,C -0.9519,E1 20.3182,E2 376.1064} C_DIS
LIN {X 31.1827,Y 121.5785,Z 146,A 73.3516,B 20.2528,C -0.9585,E1 20.3132,E2 374.2817} C_DIS
LIN {X 27.3405,Y 122.501,Z 146,A 75.0025,B 20.2531,C -0.9534,E1 20.3088,E2 372.6482} C_DIS
LIN {X 24.2401,Y 123.1523,Z 146,A 76.4252,B 20.2531,C -0.9532,E1 20.3049,E2 371.2284} C_DIS
LIN {X 21.2131,Y 123.7091,Z 146,A 77.8719,B 20.253,C -0.9554,E1 20.3009,E2 369.7773} C_DIS
LIN {X 18.4247,Y 124.1556,Z 146,A 79.2417,B 20.2528,C -0.959,E1 20.2971,E2 368.3988} C_DIS
LIN {X 15.1099,Y 124.6009,Z 146,A 80.6086,B 20.2531,C -0.9531,E1 20.2934,E2 367.0503} C_DIS
LIN {X 12.3025,Y 124.9095,Z 146,A 82.0279,B 20.2528,C -0.9585,E1 20.2894,E2 365.6168} C_DIS
LIN {X 8.6978,Y 125.2126,Z 146,A 83.7851,B 20.2526,C -0.9627,E1 20.2845,E2 363.8483} C_DIS
LIN {X 4.6219,Y 125.4288,Z 146,A 85.4906,B 20.2529,C -0.9566,E1 20.2798,E2 362.1614} C_DIS
LIN {X 0.8622,Y 125.5108,Z 146,A 87.08,B 20.2531,C -0.9515,E1 20.2754,E2 360.587} C_DIS
LIN {X -1.6429,Y 125.5037,Z 146,A 88.3931,B 20.2529,C -0.9578,E1 20.2716,E2 359.2555} C_DIS
LIN {X -4.6121,Y 125.4292,Z 146,A 89.7578,B 20.2529,C -0.9578,E1 20.2678,E2 357.8905} C_DIS
LIN {X -7.9294,Y 125.263,Z 146,A 91.1724,B 20.2531,C -0.9534,E1 20.2639,E2 356.4882} C_DIS
LIN {X -11.0227,Y 125.0295,Z 146,A 92.6202,B 20.2531,C -0.9541,E1 20.2599,E2 355.0377} C_DIS
LIN {X -13.8329,Y 124.7496,Z 146,A 93.9139,B 20.2531,C -0.9536,E1 20.2563,E2 353.7444} C_DIS
LIN {X -17.1319,Y 124.3404,Z 146,A 95.3872,B 20.2531,C -0.9511,E1 20.2522,E2 352.2771} C_DIS
LIN {X -19.9253,Y 123.9239,Z 146,A 96.8328,B 20.2529,C -0.9562,E1 20.2482,E2 350.8149} C_DIS
LIN {X -23.5353,Y 123.2871,Z 146,A 98.3324,B 20.2533,C -0.9485,E1 20.2441,E2 349.3359} C_DIS
LIN {X -26.2411,Y 122.7399,Z 146,A 99.6775,B 20.2532,C -0.9507,E1 20.2404,E2 347.9823} C_DIS
LIN {X -29.2399,Y 122.0601,Z 146,A 101.0112,B 20.2534,C -0.9468,E1 20.2368,E2 346.6575} C_DIS
LIN {X -31.9813,Y 121.371,Z 146,A 102.4055,B 20.2532,C -0.9496,E1 20.233,E2 345.2527} C_DIS
LIN {X -35.1434,Y 120.4929,Z 146,A 103.9582,B 20.2532,C -0.9501,E1 20.2289,E2 343.6952} C_DIS
LIN {X -39.3769,Y 119.1768,Z 146,A 105.9677,B 20.2533,C -0.9474,E1 20.2235,E2 341.6893} C_DIS
LIN {X -42.5148,Y 118.0935,Z 146,A 107.4261,B 20.2535,C -0.9434,E1 20.2197,E2 340.2386} C_DIS
LIN {X -45.4092,Y 117.011,Z 146,A 108.7728,B 20.2537,C -0.9393,E1 20.2162,E2 338.9004} C_DIS
LIN {X -48.0306,Y 115.9601,Z 146,A 110.1884,B 20.2536,C -0.9423,E1 20.2125,E2 337.4721} C_DIS
LIN {X -50.8572,Y 114.7487,Z 146,A 111.5408,B 20.2537,C -0.9384,E1 20.2091,E2 336.1269} C_DIS
LIN {X -53.6525,Y 113.4689,Z 146,A 112.9476,B 20.2538,C -0.9365,E1 20.2055,E2 334.7213} C_DIS
LIN {X -56.4267,Y 112.1156,Z 146,A 114.4465,B 20.2538,C -0.9377,E1 20.2017,E2 333.2139} C_DIS
LIN {X -59.1796,Y 110.6881,Z 146,A 115.7851,B 20.254,C -0.9325,E1 20.1985,E2 331.8855} C_DIS
LIN {X -62.0933,Y 109.0801,Z 146,A 117.3134,B 20.254,C -0.9303,E1 20.1947,E2 330.358} C_DIS
LIN {X -64.7456,Y 107.5271,Z 146,A 118.7211,B 20.2542,C -0.9281,E1 20.1914,E2 328.9515} C_DIS
LIN {X -67.9883,Y 105.5071,Z 146,A 120.6036,B 20.2541,C -0.9301,E1 20.1869,E2 327.0557} C_DIS
LIN {X -71.0024,Y 103.5021,Z 146,A 122.1904,B 20.2543,C -0.9245,E1 20.1832,E2 325.4783} C_DIS
LIN {X -73.5314,Y 101.721,Z 146,A 123.6116,B 20.2544,C -0.9221,E1 20.18,E2 324.0578} C_DIS
LIN {X -76.7107,Y 99.3456,Z 146,A 125.5055,B 20.2544,C -0.9215,E1 20.1758,E2 322.1572} C_DIS
LIN {X -80.212,Y 96.5407,Z 146,A 127.5992,B 20.2546,C -0.9189,E1 20.1713,E2 320.0611} C_DIS
LIN {X -83.2431,Y 93.9395,Z 146,A 129.4045,B 20.2548,C -0.9142,E1 20.1675,E2 318.2602} C_DIS
LIN {X -86.545,Y 90.9067,Z 146,A 131.4808,B 20.2549,C -0.9107,E1 20.1632,E2 316.1835} C_DIS
LIN {X -89.8235,Y 87.6689,Z 146,A 133.4686,B 20.2553,C -0.9016,E1 20.1594,E2 314.2116} C_DIS
LIN {X -92.5593,Y 84.7753,Z 146,A 135.4161,B 20.2553,C -0.9019,E1 20.1556,E2 312.2522} C_DIS
LIN {X -95.1204,Y 81.8909,Z 146,A 137.1756,B 20.2555,C -0.8975,E1 20.1524,E2 310.4955} C_DIS
LIN {X -97.9847,Y 78.442,Z 146,A 139.2674,B 20.2557,C -0.894,E1 20.1487,E2 308.4016} C_DIS
LIN {X -100.816,Y 74.7677,Z 146,A 141.2429,B 20.2561,C -0.8834,E1 20.1454,E2 306.4451} C_DIS
LIN {X -102.7617,Y 72.0705,Z 146,A 142.7744,B 20.2562,C -0.8798,E1 20.1429,E2 304.9144} C_DIS
LIN {X -104.4959,Y 69.5317,Z 146,A 144.1333,B 20.2565,C -0.8744,E1 20.1408,E2 303.5626} C_DIS
LIN {X -106.3849,Y 66.6062,Z 146,A 145.9228,B 20.2564,C -0.8773,E1 20.1381,E2 301.7533} C_DIS
LIN {X -108.4414,Y 63.203,Z 146,A 147.6758,B 20.2567,C -0.87,E1 20.1356,E2 300.0101} C_DIS
LIN {X -110.0792,Y 60.3046,Z 146,A 149.0874,B 20.257,C -0.8618,E1 20.1337,E2 298.6129} C_DIS
LIN {X -111.5467,Y 57.5441,Z 146,A 150.5577,B 20.257,C -0.8593,E1 20.1318,E2 297.14} C_DIS
LIN {X -112.9022,Y 54.8381,Z 146,A 151.98,B 20.2572,C -0.8568,E1 20.1301,E2 295.7154} C_DIS
LIN {X -114.1971,Y 52.0864,Z 146,A 153.3757,B 20.2573,C -0.853,E1 20.1284,E2 294.3209} C_DIS
LIN {X -115.464,Y 49.2141,Z 146,A 154.8193,B 20.2575,C -0.8492,E1 20.1268,E2 292.8785} C_DIS
LIN {X -116.5409,Y 46.6036,Z 146,A 156.1155,B 20.2576,C -0.8456,E1 20.1255,E2 291.5835} C_DIS
LIN {X -117.6488,Y 43.7311,Z 146,A 157.531,B 20.2578,C -0.8418,E1 20.1241,E2 290.169} C_DIS
LIN {X -118.7702,Y 40.5897,Z 146,A 159.0652,B 20.258,C -0.8376,E1 20.1227,E2 288.636} C_DIS
LIN {X -119.6524,Y 37.9074,Z 146,A 160.3773,B 20.258,C -0.8345,E1 20.1215,E2 287.3234} C_DIS
LIN {X -120.6201,Y 34.709,Z 146,A 161.899,B 20.2583,C -0.8297,E1 20.1203,E2 285.8045} C_DIS
LIN {X -121.4329,Y 31.7494,Z 146,A 163.2982,B 20.2584,C -0.8254,E1 20.1193,E2 284.4077} C_DIS
LIN {X -122.1152,Y 29.0111,Z 146,A 164.6083,B 20.2586,C -0.8222,E1 20.1185,E2 283.0972} C_DIS
LIN {X -122.9106,Y 25.4317,Z 146,A 166.1631,B 20.2589,C -0.8127,E1 20.1176,E2 281.5584} C_DIS
LIN {X -123.5396,Y 22.1719,Z 146,A 167.8686,B 20.2589,C -0.8148,E1 20.1167,E2 279.8341} C_DIS
LIN {X -124.1579,Y 18.4089,Z 146,A 169.6728,B 20.2589,C -0.8116,E1 20.1159,E2 278.0255} C_DIS
LIN {X -124.601,Y 15.1092,Z 146,A 171.046,B 20.2594,C -0.8016,E1 20.1154,E2 276.671} C_DIS
LIN {X -124.9095,Y 12.3026,Z 146,A 172.535,B 20.2592,C -0.8047,E1 20.115,E2 275.1616} C_DIS
LIN {X -125.2617,Y 7.9511,Z 146,A 174.5472,B 20.2594,C -0.7992,E1 20.1146,E2 273.1504} C_DIS
LIN {X -125.4697,Y 3.327,Z 146,A 176.6358,B 20.2597,C -0.7917,E1 20.1144,E2 271.0677} C_DIS
LIN {X -125.5186,Y -0.0004,Z 146,A 178.2112,B 20.2598,C -0.7888,E1 20.1144,E2 269.4885} C_DIS
LIN {X -125.4647,Y -3.5055,Z 146,A 179.7603,B 20.2601,C -0.7821,E1 20.1144,E2 267.9474} C_DIS
LIN {X -125.3093,Y -7.179,Z 146,A -178.47,B 20.2601,C -0.7801,E1 20.1147,E2 266.1699} C_DIS
LIN {X -125.0296,Y -11.021,Z 146,A -176.848,B 20.2605,C -0.7697,E1 20.115,E2 264.5658} C_DIS
LIN {X -124.7494,Y -13.8346,Z 146,A -175.3795,B 20.2605,C -0.7721,E1 20.1155,E2 263.0792} C_DIS
LIN {X -124.2453,Y -17.7972,Z 146,A -173.6422,B 20.2608,C -0.7634,E1 20.1161,E2 261.3542} C_DIS
LIN {X -123.6228,Y -21.707,Z 146,A -171.9554,B 20.2611,C -0.7535,E1 20.1169,E2 259.6835} C_DIS
LIN {X -123.0533,Y -24.7303,Z 146,A -170.4536,B 20.2611,C -0.7527,E1 20.1177,E2 258.1727} C_DIS
LIN {X -122.4096,Y -27.7406,Z 146,A -169.0281,B 20.2613,C -0.7492,E1 20.1186,E2 256.7468} C_DIS
LIN {X -121.7482,Y -30.514,Z 146,A -167.7276,B 20.2614,C -0.7452,E1 20.1194,E2 255.4483} C_DIS
LIN {X -120.9655,Y -33.4819,Z 146,A -166.2306,B 20.2614,C -0.7445,E1 20.1205,E2 253.9423} C_DIS
LIN {X -120.0371,Y -36.6698,Z 146,A -164.8564,B 20.2618,C -0.7349,E1 20.1216,E2 252.586} C_DIS
LIN {X -119.1779,Y -39.3737,Z 146,A -163.4227,B 20.2618,C -0.7361,E1 20.1229,E2 251.1384} C_DIS
LIN {X -118.0921,Y -42.5184,Z 146,A -161.9218,B 20.2619,C -0.7311,E1 20.1243,E2 249.6414} C_DIS
LIN {X -117.012,Y -45.4065,Z 146,A -160.4282,B 20.2619,C -0.7302,E1 20.1258,E2 248.1398} C_DIS
LIN {X -115.3607,Y -49.4531,Z 146,A -158.5287,B 20.2623,C -0.721,E1 20.1278,E2 246.2536} C_DIS
LIN {X -114.1138,Y -52.2665,Z 146,A -157.1158,B 20.2623,C -0.7174,E1 20.1294,E2 244.8414} C_DIS
LIN {X -112.7863,Y -55.073,Z 146,A -155.6939,B 20.2625,C -0.7137,E1 20.1311,E2 243.4206} C_DIS
LIN {X -111.2976,Y -58.0217,Z 146,A -154.2901,B 20.2628,C -0.7058,E1 20.1329,E2 242.0302} C_DIS
LIN {X -109.9783,Y -60.489,Z 146,A -152.8226,B 20.2627,C -0.7093,E1 20.1349,E2 240.5427} C_DIS
LIN {X -108.0369,Y -63.8919,Z 146,A -150.9181,B 20.2627,C -0.7089,E1 20.1376,E2 238.627} C_DIS
LIN {X -105.9068,Y -67.364,Z 146,A -149.2395,B 20.263,C -0.6975,E1 20.14,E2 236.9707} C_DIS
LIN {X -104.3644,Y -69.7288,Z 146,A -147.88,B 20.263,C -0.6968,E1 20.1421,E2 235.6045} C_DIS
LIN {X -102.4712,Y -72.4824,Z 146,A -146.3344,B 20.2632,C -0.6938,E1 20.1446,E2 234.058} C_DIS
LIN {X -100.6704,Y -74.9632,Z 146,A -144.8975,B 20.2632,C -0.6918,E1 20.147,E2 232.6183} C_DIS
LIN {X -98.4902,Y -77.8063,Z 146,A -143.1677,B 20.2632,C -0.6914,E1 20.15,E2 230.8792} C_DIS
LIN {X -96.0392,Y -80.8116,Z 146,A -141.4847,B 20.2635,C -0.6841,E1 20.1529,E2 229.2076} C_DIS
LIN {X -93.4278,Y -83.8169,Z 146,A -139.5795,B 20.2635,C -0.6833,E1 20.1565,E2 227.2938} C_DIS
LIN {X -90.4585,Y -87.014,Z 146,A -137.5415,B 20.2635,C -0.6807,E1 20.1604,E2 225.2522} C_DIS
LIN {X -87.6599,Y -89.8324,Z 146,A -135.8625,B 20.2639,C -0.672,E1 20.1637,E2 223.5897} C_DIS
LIN {X -84.8628,Y -92.4788,Z 146,A -134.1152,B 20.2639,C -0.6681,E1 20.1673,E2 221.8448} C_DIS
LIN {X -82.5615,Y -94.539,Z 146,A -132.5451,B 20.2639,C -0.6713,E1 20.1706,E2 220.2573} C_DIS
LIN {X -79.0105,Y -97.5266,Z 146,A -130.4246,B 20.264,C -0.6675,E1 20.1752,E2 218.1378} C_DIS
LIN {X -75.9191,Y -99.9523,Z 146,A -128.7415,B 20.2642,C -0.6601,E1 20.1788,E2 216.4683} C_DIS
LIN {X -73.5572,Y -101.7024,Z 146,A -127.3836,B 20.2642,C -0.6585,E1 20.1819,E2 215.1092} C_DIS
LIN {X -70.8016,Y -103.6399,Z 146,A -125.7597,B 20.2642,C -0.6592,E1 20.1857,E2 213.4762} C_DIS
LIN {X -67.1473,Y -106.0438,Z 146,A -123.8771,B 20.2645,C -0.6518,E1 20.19,E2 211.6075} C_DIS
LIN {X -64.5318,Y -107.6558,Z 146,A -122.4712,B 20.2645,C -0.6499,E1 20.1934,E2 210.2016} C_DIS
LIN {X -61.1665,Y -109.603,Z 146,A -120.5247,B 20.2645,C -0.6539,E1 20.1982,E2 208.2361} C_DIS
LIN {X -57.5775,Y -111.5297,Z 146,A -118.8271,B 20.2647,C -0.6453,E1 20.2023,E2 206.5575} C_DIS
LIN {X -54.825,Y -112.9087,Z 146,A -117.2615,B 20.2646,C -0.6498,E1 20.2063,E2 204.9739} C_DIS
LIN {X -52.0413,Y -114.2179,Z 146,A -115.9936,B 20.2648,C -0.6429,E1 20.2095,E2 203.7219} C_DIS
LIN {X -49.2288,Y -115.4577,Z 146,A -114.5884,B 20.2648,C -0.6415,E1 20.2131,E2 202.3166} C_DIS
LIN {X -45.757,Y -116.8758,Z 146,A -112.7482,B 20.2648,C -0.6448,E1 20.2179,E2 200.4618} C_DIS
LIN {X -42.2918,Y -118.1739,Z 146,A -111.156,B 20.2648,C -0.6395,E1 20.222,E2 198.8809} C_DIS
LIN {X -38.484,Y -119.4682,Z 146,A -109.2188,B 20.2648,C -0.642,E1 20.2272,E2 196.932} C_DIS
LIN {X -34.2315,Y -120.7559,Z 146,A -107.4447,B 20.2651,C -0.6307,E1 20.2319,E2 195.187} C_DIS
LIN {X -31.7535,Y -121.4318,Z 146,A -106.1401,B 20.2651,C -0.635,E1 20.2354,E2 193.8672} C_DIS
LIN {X -28.9971,Y -122.1186,Z 146,A -104.8428,B 20.2651,C -0.6344,E1 20.2389,E2 192.5696} C_DIS
LIN {X -25.9968,Y -122.7926,Z 146,A -103.4076,B 20.2651,C -0.6349,E1 20.2429,E2 191.1306} C_DIS
LIN {X -22.9798,Y -123.3933,Z 146,A -101.9726,B 20.265,C -0.6356,E1 20.2468,E2 189.6918} C_DIS
LIN {X -19.7025,Y -123.9584,Z 146,A -100.5928,B 20.2652,C -0.6296,E1 20.2506,E2 188.3275} C_DIS
LIN {X -16.6399,Y -124.406,Z 146,A -99.0876,B 20.2651,C -0.6329,E1 20.2548,E2 186.8112} C_DIS
LIN {X -13.837,Y -124.7492,Z 146,A -97.7954,B 20.2651,C -0.6329,E1 20.2584,E2 185.5183} C_DIS
LIN {X -10.5278,Y -125.0713,Z 146,A -96.1618,B 20.2649,C -0.6373,E1 20.2629,E2 183.8708} C_DIS
LIN {X -5.9159,Y -125.3747,Z 146,A -94.2131,B 20.2651,C -0.6309,E1 20.2683,E2 181.9399} C_DIS
LIN {X -2.8263,Y -125.4836,Z 146,A -92.7955,B 20.2651,C -0.6313,E1 20.2723,E2 180.5209} C_DIS
LIN {X 0.2421,Y -125.5143,Z 146,A -91.4333,B 20.2651,C -0.63,E1 20.2761,E2 179.1625} C_DIS
LIN {X 0.2421,Y -125.5143,Z 146,A -91.4333,B 20.2651,C -0.63,E1 20.2761,E2 179.1625} C_DIS
Enddeposition()
LIN {X 0.936,Y -131.6046,Z 147,A -92.5474,B 24.9668,C -1.3317,E1 25.002,E2 179.0325} C_DIS
Startdeposition()
$VEL.CP = VEL_PRINT
LIN {X -1.6769,Y -131.6004,Z 147,A -94.264,B 24.9683,C -1.3014,E1 24.997,E2 180.8208} C_DIS
LIN {X -5.673,Y -131.4888,Z 147,A -96.0462,B 24.9683,C -1.299,E1 24.992,E2 182.6089} C_DIS
LIN {X -9.6294,Y -131.2572,Z 147,A -97.6224,B 24.968,C -1.3067,E1 24.9877,E2 184.1675} C_DIS
LIN {X -12.8542,Y -130.981,Z 147,A -99.1609,B 24.9683,C -1.3001,E1 24.9834,E2 185.7223} C_DIS
LIN {X -17.0993,Y -130.4944,Z 147,A -100.9245,B 24.9681,C -1.3054,E1 24.9785,E2 187.4747} C_DIS
LIN {X -20.5568,Y -129.9952,Z 147,A -102.4839,B 24.9681,C -1.3038,E1 24.9742,E2 189.0392} C_DIS
LIN {X -24.6067,Y -129.2891,Z 147,A -104.2396,B 24.9681,C -1.3062,E1 24.9694,E2 190.791} C_DIS
LIN {X -28.0274,Y -128.5911,Z 147,A -105.7108,B 24.9679,C -1.3094,E1 24.9654,E2 192.2564} C_DIS
LIN {X -31.2727,Y -127.8411,Z 147,A -107.21,B 24.9679,C -1.3076,E1 24.9613,E2 193.7618} C_DIS
LIN {X -35.1781,Y -126.8215,Z 147,A -109.1985,B 24.9685,C -1.2971,E1 24.9558,E2 195.7783} C_DIS
LIN {X -40.111,Y -125.3484,Z 147,A -111.2112,B 24.9678,C -1.3103,E1 24.9505,E2 197.7632} C_DIS
LIN {X -43.1786,Y -124.325,Z 147,A -112.6218,B 24.9678,C -1.3113,E1 24.9468,E2 199.174} C_DIS
LIN {X -46.3368,Y -123.1829,Z 147,A -114.055,B 24.9677,C -1.3141,E1 24.9431,E2 200.6035} C_DIS
LIN {X -49.4658,Y -121.9602,Z 147,A -115.5496,B 24.9677,C -1.314,E1 24.9392,E2 202.1017} C_DIS
LIN {X -52.3703,Y -120.7412,Z 147,A -116.9368,B 24.9677,C -1.3147,E1 24.9356,E2 203.4905} C_DIS
LIN {X -55.3676,Y -119.3965,Z 147,A -118.3698,B 24.9676,C -1.3162,E1 24.932,E2 204.9234} C_DIS
LIN {X -58.4913,Y -117.8979,Z 147,A -119.8934,B 24.9675,C -1.3173,E1 24.9281,E2 206.4483} C_DIS
LIN {X -61.77,Y -116.2151,Z 147,A -121.5453,B 24.9675,C -1.317,E1 24.924,E2 208.1053} C_DIS
LIN {X -65.5406,Y -114.1321,Z 147,A -123.3425,B 24.9672,C -1.3236,E1 24.9197,E2 209.8923} C_DIS
LIN {X -68.7063,Y -112.2543,Z 147,A -125.0674,B 24.9674,C -1.3199,E1 24.9155,E2 211.6312} C_DIS
LIN {X -72.6,Y -109.7765,Z 147,A -127.1084,B 24.9673,C -1.3216,E1 24.9107,E2 213.6748} C_DIS
LIN {X -76.2666,Y -107.2618,Z 147,A -129.0585,B 24.9672,C -1.3241,E1 24.9063,E2 215.6255} C_DIS
LIN {X -79.8814,Y -104.597,Z 147,A -130.9895,B 24.9669,C -1.3288,E1 24.902,E2 217.5522} C_DIS
LIN {X -83.4843,Y -101.7448,Z 147,A -132.9746,B 24.9667,C -1.3334,E1 24.8977,E2 219.534} C_DIS
LIN {X -86.8427,Y -98.8943,Z 147,A -134.9456,B 24.9667,C -1.3346,E1 24.8935,E2 221.5099} C_DIS
LIN {X -90.1129,Y -95.9235,Z 147,A -136.8863,B 24.9665,C -1.3377,E1 24.8895,E2 223.4509} C_DIS
LIN {X -93.3534,Y -92.7723,Z 147,A -138.8244,B 24.9662,C -1.3434,E1 24.8857,E2 225.3836} C_DIS
LIN {X -95.549,Y -90.5098,Z 147,A -140.14,B 24.9659,C -1.3492,E1 24.8831,E2 226.6911} C_DIS
LIN {X -98.3244,Y -87.4874,Z 147,A -142.0382,B 24.9659,C -1.3479,E1 24.8796,E2 228.6009} C_DIS
LIN {X -100.9898,Y -84.396,Z 147,A -143.8079,B 24.9657,C -1.3525,E1 24.8764,E2 230.3678} C_DIS
LIN {X -103.8023,Y -80.9122,Z 147,A -145.745,B 24.9655,C -1.3578,E1 24.873,E2 232.3013} C_DIS
LIN {X -106.3647,Y -77.5128,Z 147,A -147.6527,B 24.9654,C -1.3599,E1 24.8698,E2 234.2133} C_DIS
LIN {X -108.8493,Y -73.9829,Z 147,A -149.4922,B 24.965,C -1.3666,E1 24.8669,E2 236.0458} C_DIS
LIN {X -111.2219,Y -70.3652,Z 147,A -151.3974,B 24.9648,C -1.3706,E1 24.864,E2 237.9512} C_DIS
LIN {X -113.6162,Y -66.4304,Z 147,A -153.4286,B 24.9646,C -1.3748,E1 24.8611,E2 239.9828} C_DIS
LIN {X -115.7872,Y -62.5699,Z 147,A -155.3503,B 24.9643,C -1.3805,E1 24.8585,E2 241.9012} C_DIS
LIN {X -117.3232,Y -59.6349,Z 147,A -156.7221,B 24.9639,C -1.3879,E1 24.8568,E2 243.2625} C_DIS
LIN {X -118.7829,Y -56.6718,Z 147,A -158.1726,B 24.9637,C -1.3915,E1 24.855,E2 244.7124} C_DIS
LIN {X -120.1825,Y -53.64,Z 147,A -159.6435,B 24.9636,C -1.3949,E1 24.8533,E2 246.1833} C_DIS
LIN {X -121.5188,Y -50.5401,Z 147,A -161.0912,B 24.9633,C -1.4003,E1 24.8518,E2 247.6262} C_DIS
LIN {X -122.7938,Y -47.3591,Z 147,A -162.5469,B 24.9629,C -1.4064,E1 24.8503,E2 249.0752} C_DIS
LIN {X -123.8712,Y -44.4641,Z 147,A -164.0088,B 24.963,C -1.4049,E1 24.8489,E2 250.5491} C_DIS
LIN {X -125.2516,Y -40.414,Z 147,A -165.8912,B 24.9628,C -1.4097,E1 24.8472,E2 252.4308} C_DIS
LIN {X -126.3166,Y -36.9491,Z 147,A -167.3989,B 24.9623,C -1.4179,E1 24.846,E2 253.9276} C_DIS
LIN {X -127.2255,Y -33.6874,Z 147,A -168.8945,B 24.9621,C -1.4215,E1 24.8449,E2 255.4234} C_DIS
LIN {X -128.1522,Y -29.977,Z 147,A -170.6847,B 24.9621,C -1.4208,E1 24.8437,E2 257.2258} C_DIS
LIN {X -128.9774,Y -26.191,Z 147,A -172.2404,B 24.9616,C -1.4324,E1 24.8428,E2 258.763} C_DIS
LIN {X -129.6096,Y -22.8607,Z 147,A -173.8205,B 24.9616,C -1.4322,E1 24.842,E2 260.353} C_DIS
LIN {X -130.27,Y -18.7325,Z 147,A -175.6005,B 24.9612,C -1.4399,E1 24.8413,E2 262.1251} C_DIS
LIN {X -130.7201,Y -15.2817,Z 147,A -177.1973,B 24.9612,C -1.441,E1 24.8407,E2 263.7289} C_DIS
LIN {X -131.1602,Y -10.8732,Z 147,A -179.048,B 24.9606,C -1.451,E1 24.8403,E2 265.5669} C_DIS
LIN {X -131.4267,Y -6.9534,Z 147,A 179.1509,B 24.9605,C -1.4523,E1 24.84,E2 267.3757} C_DIS
LIN {X -131.5749,Y -3.092,Z 147,A 177.3479,B 24.9605,C -1.4521,E1 24.8398,E2 269.19} C_DIS
LIN {X -131.5859,Y 2.5459,Z 147,A 174.9472,B 24.9599,C -1.4628,E1 24.8398,E2 271.5798} C_DIS
LIN {X -131.4724,Y 6.043,Z 147,A 173.4331,B 24.9596,C -1.4682,E1 24.84,E2 273.09} C_DIS
LIN {X -131.0874,Y 11.7354,Z 147,A 171.1371,B 24.9587,C -1.4852,E1 24.8405,E2 275.3593} C_DIS
LIN {X -130.3868,Y 17.915,Z 147,A 168.3398,B 24.9584,C -1.4899,E1 24.8414,E2 278.1621} C_DIS
LIN {X -129.6428,Y 22.675,Z 147,A 165.8208,B 24.9591,C -1.477,E1 24.8426,E2 280.7269} C_DIS
LIN {X -129.007,Y 26.0454,Z 147,A 164.813,B 24.9576,C -1.5047,E1 24.8431,E2 281.6745} C_DIS
LIN {X -128.0595,Y 30.3665,Z 147,A 162.7881,B 24.9575,C -1.5063,E1 24.8443,E2 283.7077} C_DIS
LIN {X -127.2246,Y 33.6909,Z 147,A 161.216,B 24.9575,C -1.5074,E1 24.8454,E2 285.2863} C_DIS
LIN {X -126.3043,Y 36.9909,Z 147,A 159.7107,B 24.9572,C -1.5115,E1 24.8466,E2 286.7904} C_DIS
LIN {X -125.3246,Y 40.1853,Z 147,A 158.2824,B 24.9569,C -1.5175,E1 24.8478,E2 288.2128} C_DIS
LIN {X -124.2839,Y 43.2971,Z 147,A 156.8616,B 24.9566,C -1.5224,E1 24.849,E2 289.63} C_DIS
LIN {X -123.2072,Y 46.2718,Z 147,A 155.4467,B 24.9564,C -1.5249,E1 24.8504,E2 291.0467} C_DIS
LIN {X -122.0053,Y 49.3539,Z 147,A 154.0081,B 24.9562,C -1.5295,E1 24.8519,E2 292.4824} C_DIS
LIN {X -120.7231,Y 52.4122,Z 147,A 152.5412,B 24.956,C -1.5329,E1 24.8535,E2 293.9494} C_DIS
LIN {X -119.3938,Y 55.3734,Z 147,A 151.095,B 24.9558,C -1.5357,E1 24.8552,E2 295.3969} C_DIS
LIN {X -117.9604,Y 58.3646,Z 147,A 149.6542,B 24.9556,C -1.5403,E1 24.8569,E2 296.8346} C_DIS
LIN {X -116.4815,Y 61.2628,Z 147,A 148.284,B 24.9552,C -1.5468,E1 24.8587,E2 298.1967} C_DIS
LIN {X -114.5412,Y 64.8231,Z 147,A 146.3246,B 24.9554,C -1.5428,E1 24.8613,E2 300.1759} C_DIS
LIN {X -112.2838,Y 68.6582,Z 147,A 144.4013,B 24.955,C -1.5491,E1 24.8641,E2 302.094} C_DIS
LIN {X -108.7863,Y 74.0759,Z 147,A 141.5664,B 24.9546,C -1.5558,E1 24.8685,E2 304.9271} C_DIS
LIN {X -106.2432,Y 77.6791,Z 147,A 139.6256,B 24.9544,C -1.5602,E1 24.8716,E2 306.8669} C_DIS
LIN {X -103.457,Y 81.3524,Z 147,A 137.625,B 24.9541,C -1.566,E1 24.875,E2 308.8633} C_DIS
LIN {X -100.8648,Y 84.545,Z 147,A 135.8365,B 24.9538,C -1.5709,E1 24.8782,E2 310.6484} C_DIS
LIN {X -98.0881,Y 87.7514,Z 147,A 133.9795,B 24.9535,C -1.5752,E1 24.8816,E2 312.5035} C_DIS
LIN {X -95.4025,Y 90.6646,Z 147,A 132.2394,B 24.9533,C -1.5789,E1 24.8849,E2 314.2425} C_DIS
LIN {X -92.3395,Y 93.7819,Z 147,A 130.3327,B 24.953,C -1.5834,E1 24.8887,E2 316.1466} C_DIS
LIN {X -89.2142,Y 96.7597,Z 147,A 128.4465,B 24.9528,C -1.5876,E1 24.8925,E2 318.0306} C_DIS
LIN {X -85.8998,Y 99.7135,Z 147,A 126.5159,B 24.9525,C -1.5922,E1 24.8966,E2 319.9578} C_DIS
LIN {X -82.4903,Y 102.5521,Z 147,A 124.5925,B 24.9522,C -1.5969,E1 24.9007,E2 321.8773} C_DIS
LIN {X -79.0315,Y 105.2411,Z 147,A 122.7033,B 24.9519,C -1.6019,E1 24.9049,E2 323.7615} C_DIS
LIN {X -76.1009,Y 107.3792,Z 147,A 120.7668,B 24.9528,C -1.588,E1 24.9094,E2 325.7378} C_DIS
LIN {X -73.0952,Y 109.447,Z 147,A 119.6811,B 24.9511,C -1.6154,E1 24.9118,E2 326.7618} C_DIS
LIN {X -70.3335,Y 111.242,Z 147,A 118.0207,B 24.9516,C -1.6072,E1 24.9157,E2 328.447} C_DIS
LIN {X -66.4129,Y 113.6265,Z 147,A 116.0258,B 24.9514,C -1.611,E1 24.9205,E2 330.4389} C_DIS
LIN {X -62.6315,Y 115.7541,Z 147,A 114.0978,B 24.9513,C -1.6125,E1 24.9252,E2 332.3691} C_DIS
LIN {X -59.498,Y 117.3929,Z 147,A 112.6511,B 24.9508,C -1.6196,E1 24.9288,E2 333.8027} C_DIS
LIN {X -56.4966,Y 118.8666,Z 147,A 111.2093,B 24.9507,C -1.6226,E1 24.9324,E2 335.241} C_DIS
LIN {X -52.9831,Y 120.4763,Z 147,A 109.3795,B 24.9509,C -1.618,E1 24.9371,E2 337.0863} C_DIS
LIN {X -49.1393,Y 122.0918,Z 147,A 107.7129,B 24.9503,C -1.6279,E1 24.9413,E2 338.7331} C_DIS
LIN {X -46.0595,Y 123.2867,Z 147,A 106.2796,B 24.9503,C -1.6301,E1 24.9451,E2 340.1642} C_DIS
LIN {X -42.9103,Y 124.418,Z 147,A 104.7875,B 24.9503,C -1.6302,E1 24.949,E2 341.6589} C_DIS
LIN {X -39.9056,Y 125.414,Z 147,A 103.4669,B 24.9499,C -1.6347,E1 24.9525,E2 342.9713} C_DIS
LIN {X -36.944,Y 126.318,Z 147,A 102.0392,B 24.9501,C -1.6323,E1 24.9563,E2 344.4071} C_DIS
LIN {X -33.1594,Y 127.3663,Z 147,A 100.2062,B 24.9503,C -1.628,E1 24.9613,E2 346.2532} C_DIS
LIN {X -29.3839,Y 128.2876,Z 147,A 98.6584,B 24.9498,C -1.6367,E1 24.9655,E2 347.7823} C_DIS
LIN {X -26.2062,Y 128.9743,Z 147,A 97.2408,B 24.9498,C -1.6378,E1 24.9693,E2 349.1989} C_DIS
LIN {X -22.5594,Y 129.6635,Z 147,A 95.347,B 24.9505,C -1.6253,E1 24.9746,E2 351.1244} C_DIS
LIN {X -18.3003,Y 130.3317,Z 147,A 93.4895,B 24.9504,C -1.6275,E1 24.9798,E2 352.9781} C_DIS
LIN {X -14.2055,Y 130.8411,Z 147,A 91.9221,B 24.9496,C -1.6399,E1 24.984,E2 354.5171} C_DIS
LIN {X -10.403,Y 131.1999,Z 147,A 90.1443,B 24.9499,C -1.635,E1 24.989,E2 356.3075} C_DIS
LIN {X -6.3161,Y 131.4587,Z 147,A 88.3878,B 24.9498,C -1.637,E1 24.9939,E2 358.0599} C_DIS
LIN {X -2.1411,Y 131.5927,Z 147,A 86.6526,B 24.9495,C -1.6416,E1 24.9987,E2 359.784} C_DIS
LIN {X 1.9927,Y 131.5951,Z 147,A 84.8592,B 24.9495,C -1.6423,E1 25.0037,E2 361.5758} C_DIS
LIN {X 5.7929,Y 131.4842,Z 147,A 83.0813,B 24.9498,C -1.6362,E1 25.0087,E2 363.3677} C_DIS
LIN {X 9.8109,Y 131.244,Z 147,A 81.5004,B 24.9493,C -1.6448,E1 25.0131,E2 364.9275} C_DIS
LIN {X 13.4441,Y 130.923,Z 147,A 79.7834,B 24.9497,C -1.6381,E1 25.0179,E2 366.6594} C_DIS
LIN {X 17.0993,Y 130.4944,Z 147,A 78.2627,B 24.9495,C -1.6419,E1 25.0221,E2 368.1698} C_DIS
LIN {X 20.6123,Y 129.9866,Z 147,A 76.615,B 24.9498,C -1.6362,E1 25.0266,E2 369.8295} C_DIS
LIN {X 24.8366,Y 129.2451,Z 147,A 74.9296,B 24.9493,C -1.6447,E1 25.0312,E2 371.4928} C_DIS
LIN {X 30.8166,Y 127.951,Z 147,A 71.6293,B 24.9514,C -1.6109,E1 25.0404,E2 374.8687} C_DIS
LIN {X 35.3299,Y 126.779,Z 147,A 70.1315,B 24.9498,C -1.6366,E1 25.0443,E2 376.3031} C_DIS
LIN {X 38.5785,Y 125.8285,Z 147,A 68.6837,B 24.9498,C -1.6368,E1 25.0481,E2 377.748} C_DIS
LIN {X 41.7318,Y 124.8182,Z 147,A 67.2852,B 24.9498,C -1.6379,E1 25.0518,E2 379.1414} C_DIS
LIN {X 44.9044,Y 123.7124,Z 147,A 65.8397,B 24.9498,C -1.6374,E1 25.0556,E2 380.5851} C_DIS
LIN {X 48.0006,Y 122.5444,Z 147,A 64.3784,B 24.9499,C -1.6349,E1 25.0594,E2 382.0492} C_DIS
LIN {X 50.8684,Y 121.3816,Z 147,A 63.0139,B 24.9501,C -1.6325,E1 25.063,E2 383.416} C_DIS
LIN {X 53.7918,Y 120.1146,Z 147,A 61.6917,B 24.9499,C -1.6343,E1 25.0663,E2 384.7307} C_DIS
LIN {X 62.9293,Y 115.5919,Z 147,A 57.348,B 24.95,C -1.6334,E1 25.0772,E2 389.0649} C_DIS
LIN {X 65.7158,Y 114.031,Z 147,A 55.7136,B 24.9509,C -1.6186,E1 25.0812,E2 390.7295} C_DIS
LIN {X 69.4911,Y 111.7701,Z 147,A 53.831,B 24.9509,C -1.6174,E1 25.0857,E2 392.609} C_DIS
LIN {X 73.3068,Y 109.3058,Z 147,A 51.0379,B 24.9537,C -1.5717,E1 25.0924,E2 395.5007} C_DIS
LIN {X 78.5239,Y 105.6199,Z 147,A 49.4692,B 24.9502,C -1.63,E1 25.0956,E2 396.926} C_DIS
LIN {X 82.0391,Y 102.9134,Z 147,A 47.1589,B 24.9516,C -1.6064,E1 25.1008,E2 399.2836} C_DIS
LIN {X 85.546,Y 100.018,Z 147,A 45.1991,B 24.9518,C -1.6036,E1 25.105,E2 401.2426} C_DIS
LIN {X 88.6578,Y 97.27,Z 147,A 43.3953,B 24.952,C -1.6001,E1 25.1087,E2 403.0475} C_DIS
LIN {X 91.8391,Y 94.2725,Z 147,A 41.4776,B 24.9523,C -1.5952,E1 25.1126,E2 404.9687} C_DIS
LIN {X 94.9483,Y 91.1398,Z 147,A 39.5589,B 24.9526,C -1.5911,E1 25.1164,E2 406.8888} C_DIS
LIN {X 98.0285,Y 87.8179,Z 147,A 37.6302,B 24.9526,C -1.5889,E1 25.12,E2 408.8143} C_DIS
LIN {X 101.0007,Y 84.3831,Z 147,A 35.6944,B 24.9528,C -1.5864,E1 25.1235,E2 410.7472} C_DIS
LIN {X 103.7172,Y 81.0211,Z 147,A 33.7999,B 24.9532,C -1.5811,E1 25.1268,E2 412.6453} C_DIS
LIN {X 106.3238,Y 77.5692,Z 147,A 31.866,B 24.9536,C -1.5736,E1 25.13,E2 414.5876} C_DIS
LIN {X 108.8101,Y 74.0407,Z 147,A 30.0228,B 24.9538,C -1.5706,E1 25.133,E2 416.4287} C_DIS
LIN {X 111.2004,Y 70.3993,Z 147,A 28.152,B 24.954,C -1.567,E1 25.1358,E2 418.2988} C_DIS
LIN {X 113.4087,Y 66.7837,Z 147,A 26.2723,B 24.9544,C -1.56,E1 25.1385,E2 420.1852} C_DIS
LIN {X 115.6666,Y 62.7923,Z 147,A 24.3339,B 24.9545,C -1.5576,E1 25.1411,E2 422.1193} C_DIS
LIN {X 117.3303,Y 59.6211,Z 147,A 22.8785,B 24.9545,C -1.5588,E1 25.143,E2 423.5641} C_DIS
LIN {X 118.805,Y 56.6255,Z 147,A 21.4237,B 24.9547,C -1.5545,E1 25.1447,E2 425.0212} C_DIS
LIN {X 120.2103,Y 53.5777,Z 147,A 19.9828,B 24.9549,C -1.5513,E1 25.1464,E2 426.4618} C_DIS
LIN {X 121.5585,Y 50.4449,Z 147,A 18.5579,B 24.9549,C -1.5502,E1 25.1479,E2 427.8816} C_DIS
LIN {X 122.664,Y 47.6929,Z 147,A 17.2362,B 24.9553,C -1.5447,E1 25.1493,E2 429.209} C_DIS
LIN {X 123.8496,Y 44.5239,Z 147,A 15.7469,B 24.9556,C -1.5393,E1 25.1507,E2 430.7025} C_DIS
LIN {X 124.8999,Y 41.4863,Z 147,A 14.384,B 24.9557,C -1.537,E1 25.152,E2 432.0632} C_DIS
LIN {X 125.9259,Y 38.2602,Z 147,A 12.9355,B 24.9559,C -1.5338,E1 25.1532,E2 433.511} C_DIS
LIN {X 126.851,Y 35.0727,Z 147,A 11.3426,B 24.9566,C -1.5213,E1 25.1544,E2 435.1244} C_DIS
LIN {X 127.9408,Y 30.859,Z 147,A 9.603,B 24.9566,C -1.5237,E1 25.1556,E2 436.8481} C_DIS
LIN {X 128.6693,Y 27.6649,Z 147,A 8.1702,B 24.9568,C -1.5188,E1 25.1564,E2 438.284} C_DIS
LIN {X 129.3261,Y 24.413,Z 147,A 6.6751,B 24.9572,C -1.5114,E1 25.1572,E2 439.7878} C_DIS
LIN {X 130.0393,Y 20.2718,Z 147,A 4.9093,B 24.9573,C -1.509,E1 25.158,E2 441.549} C_DIS
LIN {X 130.5445,Y 16.7165,Z 147,A 3.2715,B 24.9579,C -1.4999,E1 25.1587,E2 443.1988} C_DIS
LIN {X 131.011,Y 12.5422,Z 147,A 1.5354,B 24.9579,C -1.4989,E1 25.1592,E2 444.9268} C_DIS
LIN {X 131.3406,Y 8.4223,Z 147,A -0.2765,B 24.9583,C -1.4924,E1 25.1595,E2 446.7434} C_DIS
LIN {X 131.5232,Y 4.791,Z 147,A -1.9308,B 24.9588,C -1.4832,E1 25.1597,E2 448.4093} C_DIS
LIN {X 131.6101,Y 0.5573,Z 147,A -3.5757,B 24.9585,C -1.488,E1 25.1597,E2 450.0333} C_DIS
LIN {X 131.5778,Y -2.9885,Z 147,A -5.2903,B 24.9593,C -1.4735,E1 25.1597,E2 451.7717} C_DIS
LIN {X 131.4278,Y -6.9314,Z 147,A -6.9586,B 24.9595,C -1.4706,E1 25.1595,E2 453.4371} C_DIS
LIN {X 131.1516,Y -10.9744,Z 147,A -8.648,B 24.9595,C -1.4688,E1 25.1591,E2 455.1206} C_DIS
LIN {X 130.8398,Y -14.2179,Z 147,A -10.0619,B 24.9598,C -1.4644,E1 25.1587,E2 456.5366} C_DIS
LIN {X 130.326,Y -18.3402,Z 147,A -11.8646,B 24.9601,C -1.4587,E1 25.1581,E2 458.342} C_DIS
LIN {X 129.7796,Y -21.8738,Z 147,A -13.3446,B 24.9601,C -1.4578,E1 25.1574,E2 459.8156} C_DIS
LIN {X 129.205,Y -25.0463,Z 147,A -14.9015,B 24.9609,C -1.4448,E1 25.1566,E2 461.3939} C_DIS
LIN {X 128.3254,Y -29.2184,Z 147,A -16.6732,B 24.9609,C -1.4433,E1 25.1556,E2 463.1587} C_DIS
LIN {X 126.5763,Y -36.0549,Z 147,A -20.4357,B 24.9635,C -1.3959,E1 25.1527,E2 467.0113} C_DIS
LIN {X 124.9294,Y -41.3977,Z 147,A -21.8365,B 24.9609,C -1.4442,E1 25.1517,E2 468.2904} C_DIS
LIN {X 123.8041,Y -44.6501,Z 147,A -23.6046,B 24.962,C -1.4247,E1 25.15,E2 470.0947} C_DIS
LIN {X 122.6093,Y -47.8338,Z 147,A -25.031,B 24.962,C -1.4229,E1 25.1486,E2 471.5172} C_DIS
LIN {X 121.3396,Y -50.9691,Z 147,A -26.5159,B 24.9624,C -1.4176,E1 25.147,E2 473.0065} C_DIS
LIN {X 120.0898,Y -53.8471,Z 147,A -27.8645,B 24.9625,C -1.4143,E1 25.1455,E2 474.3554} C_DIS
LIN {X 118.6582,Y -56.9328,Z 147,A -29.3532,B 24.9628,C -1.4093,E1 25.1437,E2 475.8479} C_DIS
LIN {X 116.8889,Y -60.4869,Z 147,A -31.1848,B 24.9634,C -1.3984,E1 25.1414,E2 477.6955} C_DIS
LIN {X 114.7167,Y -64.5108,Z 147,A -33.0964,B 24.9634,C -1.3967,E1 25.1388,E2 479.6011} C_DIS
LIN {X 112.5727,Y -68.1832,Z 147,A -34.9655,B 24.9638,C -1.3903,E1 25.1361,E2 481.4758} C_DIS
LIN {X 110.1673,Y -72.0062,Z 147,A -36.9603,B 24.9642,C -1.383,E1 25.1331,E2 483.4777} C_DIS
LIN {X 107.6668,Y -75.6932,Z 147,A -39.3732,B 24.9658,C -1.352,E1 25.1292,E2 485.9519} C_DIS
LIN {X 104.7692,Y -79.6563,Z 147,A -41.2472,B 24.9653,C -1.3602,E1 25.126,E2 487.7977} C_DIS
LIN {X 102.5743,Y -82.4628,Z 147,A -42.5289,B 24.9648,C -1.3705,E1 25.1239,E2 489.0491} C_DIS
LIN {X 99.9405,Y -85.6363,Z 147,A -44.3158,B 24.965,C -1.3661,E1 25.1206,E2 490.838} C_DIS
LIN {X 97.1317,Y -88.8095,Z 147,A -46.1629,B 24.9653,C -1.3612,E1 25.1172,E2 492.6886} C_DIS
LIN {X 94.0723,Y -92.0434,Z 147,A -48.0463,B 24.9653,C -1.3592,E1 25.1135,E2 494.5685} C_DIS
LIN {X 91.054,Y -95.0303,Z 147,A -49.8931,B 24.9656,C -1.3548,E1 25.1098,E2 496.4181} C_DIS
LIN {X 87.8214,Y -98.0253,Z 147,A -51.804,B 24.9658,C -1.3506,E1 25.1059,E2 498.3311} C_DIS
LIN {X 84.6688,Y -100.7609,Z 147,A -53.6225,B 24.9661,C -1.3463,E1 25.102,E2 500.1527} C_DIS
LIN {X 81.1131,Y -103.645,Z 147,A -55.6165,B 24.9663,C -1.3418,E1 25.0977,E2 502.1499} C_DIS
LIN {X 77.5459,Y -106.3407,Z 147,A -57.5696,B 24.9665,C -1.3372,E1 25.0933,E2 504.1068} C_DIS
LIN {X 74.0591,Y -108.7977,Z 147,A -59.4266,B 24.9667,C -1.3334,E1 25.089,E2 505.9665} C_DIS
LIN {X 70.2591,Y -111.2889,Z 147,A -61.3404,B 24.9667,C -1.3329,E1 25.0845,E2 507.8752} C_DIS
LIN {X 66.4041,Y -113.6317,Z 147,A -63.3211,B 24.967,C -1.3283,E1 25.0798,E2 509.8607} C_DIS
LIN {X 62.5782,Y -115.7827,Z 147,A -65.2221,B 24.9671,C -1.3253,E1 25.0751,E2 511.763} C_DIS
LIN {X 59.3928,Y -117.4465,Z 147,A -66.6449,B 24.9669,C -1.3302,E1 25.0716,E2 513.1704} C_DIS
LIN {X 56.4509,Y -118.8884,Z 147,A -68.0857,B 24.967,C -1.3271,E1 25.068,E2 514.6148} C_DIS
LIN {X 53.562,Y -120.2174,Z 147,A -69.5077,B 24.9672,C -1.3229,E1 25.0644,E2 516.0431} C_DIS
LIN {X 50.4043,Y -121.5755,Z 147,A -70.9675,B 24.9672,C -1.3226,E1 25.0606,E2 517.5002} C_DIS
LIN {X 47.4845,Y -122.7451,Z 147,A -72.3275,B 24.9673,C -1.3212,E1 25.0571,E2 518.8606} C_DIS
LIN {X 44.2119,Y -123.9621,Z 147,A -73.9778,B 24.9677,C -1.3122,E1 25.0527,E2 520.5286} C_DIS
LIN {X 40.1214,Y -125.345,Z 147,A -75.7352,B 24.9675,C -1.3163,E1 25.0481,E2 522.2729} C_DIS
LIN {X 36.6553,Y -126.4026,Z 147,A -77.2997,B 24.9676,C -1.3152,E1 25.0439,E2 523.8375} C_DIS
LIN {X 33.6625,Y -127.2321,Z 147,A -78.6268,B 24.9676,C -1.315,E1 25.0403,E2 525.1628} C_DIS
LIN {X 30.4441,Y -128.0408,Z 147,A -80.1049,B 24.9678,C -1.3118,E1 25.0363,E2 526.6464} C_DIS
LIN {X 26.3793,Y -128.9391,Z 147,A -81.8906,B 24.9678,C -1.3115,E1 25.0314,E2 528.4304} C_DIS
LIN {X 23.1423,Y -129.5592,Z 147,A -83.3399,B 24.9678,C -1.3096,E1 25.0274,E2 529.8827} C_DIS
LIN {X 19.3461,Y -130.1823,Z 147,A -85.1537,B 24.9683,C -1.301,E1 25.0224,E2 531.7149} C_DIS
LIN {X 15.4766,Y -130.6968,Z 147,A -86.6697,B 24.9679,C -1.3095,E1 25.0182,E2 533.2097} C_DIS
LIN {X 12.2999,Y -131.0342,Z 147,A -88.1484,B 24.9681,C -1.3042,E1 25.0141,E2 534.7001} C_DIS
LIN {X 8.2638,Y -131.3504,Z 147,A -89.8733,B 24.9681,C -1.3053,E1 25.0093,E2 536.4215} C_DIS
LIN {X 4.5304,Y -131.5334,Z 147,A -91.6256,B 24.9684,C -1.2982,E1 25.0044,E2 538.1901} C_DIS
LIN {X 0.936,Y -131.6046,Z 147,A -92.5463,B 24.9668,C -1.3312,E1 25.002,E2 539.0325} C_DIS
Enddeposition()
LIN {X 0.936,Y -131.6046,Z 147,A -92.5463,B 24.9668,C -1.3312,E1 25.002,E2 539.0325} C_DIS
Startdeposition()
$VEL.CP = VEL_PRINT
LIN {X 1.9706,Y -130.6409,Z 147,A -91.9507,B 24.9656,C -1.3553,E1 25.0038,E2 538.38} C_DIS
LIN {X 5.8247,Y -130.5277,Z 147,A -90.165,B 24.9653,C -1.3608,E1 25.0089,E2 536.5817} C_DIS
LIN {X 9.5558,Y -130.3056,Z 147,A -88.6516,B 24.9656,C -1.355,E1 25.013,E2 535.0827} C_DIS
LIN {X 13.2313,Y -129.9859,Z 147,A -87.0636,B 24.9656,C -1.3543,E1 25.0174,E2 533.4973} C_DIS
LIN {X 16.2263,Y -129.6461,Z 147,A -85.667,B 24.9654,C -1.359,E1 25.0213,E2 532.0906} C_DIS
LIN {X 19.2365,Y -129.2338,Z 147,A -84.4088,B 24.9656,C -1.3561,E1 25.0248,E2 530.8405} C_DIS
LIN {X 22.7536,Y -128.6591,Z 147,A -82.8064,B 24.9654,C -1.3594,E1 25.0292,E2 529.2318} C_DIS
LIN {X 25.5106,Y -128.1418,Z 147,A -81.6159,B 24.9654,C -1.3584,E1 25.0325,E2 528.0452} C_DIS
LIN {X 28.3334,Y -127.5485,Z 147,A -80.1941,B 24.965,C -1.3678,E1 25.0364,E2 526.603} C_DIS
LIN {X 31.969,Y -126.6839,Z 147,A -78.7753,B 24.9655,C -1.3579,E1 25.0402,E2 525.2096} C_DIS
LIN {X 34.8292,Y -125.9279,Z 147,A -77.3789,B 24.9651,C -1.3645,E1 25.044,E2 523.7999} C_DIS
LIN {X 37.6935,Y -125.1012,Z 147,A -76.0965,B 24.9651,C -1.3647,E1 25.0474,E2 522.5193} C_DIS
LIN {X 40.9244,Y -124.081,Z 147,A -74.6091,B 24.9651,C -1.3666,E1 25.0514,E2 521.03} C_DIS
LIN {X 44.0261,Y -123.0144,Z 147,A -73.2017,B 24.9651,C -1.3669,E1 25.0551,E2 519.6248} C_DIS
LIN {X 46.7057,Y -122.0237,Z 147,A -71.9913,B 24.9651,C -1.3663,E1 25.0582,E2 518.4184} C_DIS
LIN {X 49.6004,Y -120.8768,Z 147,A -70.5779,B 24.9648,C -1.3709,E1 25.0619,E2 516.9975} C_DIS
LIN {X 52.8144,Y -119.5062,Z 147,A -69.1404,B 24.9649,C -1.3682,E1 25.0656,E2 515.5697} C_DIS
LIN {X 55.9024,Y -118.0926,Z 147,A -67.5754,B 24.9646,C -1.3746,E1 25.0696,E2 513.9935} C_DIS
LIN {X 58.9929,Y -116.579,Z 147,A -66.1193,B 24.9646,C -1.3743,E1 25.0732,E2 512.542} C_DIS
LIN {X 62.2029,Y -114.9008,Z 147,A -64.3289,B 24.9639,C -1.3879,E1 25.0777,E2 510.7247} C_DIS
LIN {X 65.923,Y -112.8073,Z 147,A -62.6081,B 24.9642,C -1.3832,E1 25.0818,E2 509.02} C_DIS
LIN {X 69.3725,Y -110.7197,Z 147,A -60.8442,B 24.964,C -1.3864,E1 25.086,E2 507.2541} C_DIS
LIN {X 72.2961,Y -108.8329,Z 147,A -59.2093,B 24.9635,C -1.3953,E1 25.0898,E2 505.6036} C_DIS
LIN {X 75.8144,Y -106.4117,Z 147,A -57.3457,B 24.9634,C -1.3987,E1 25.0941,E2 503.7384} C_DIS
LIN {X 79.3283,Y -103.8184,Z 147,A -55.4749,B 24.9633,C -1.4005,E1 25.0983,E2 501.8702} C_DIS
LIN {X 82.4469,Y -101.3599,Z 147,A -53.7017,B 24.963,C -1.4061,E1 25.1022,E2 500.0903} C_DIS
LIN {X 85.6772,Y -98.6445,Z 147,A -51.8595,B 24.9628,C -1.41,E1 25.1061,E2 498.2462} C_DIS
LIN {X 88.9849,Y -95.6709,Z 147,A -49.9535,B 24.9626,C -1.4123,E1 25.11,E2 496.3426} C_DIS
LIN {X 91.789,Y -92.9849,Z 147,A -48.3085,B 24.9626,C -1.4133,E1 25.1133,E2 494.702} C_DIS
LIN {X 94.6655,Y -90.0542,Z 147,A -46.4796,B 24.9623,C -1.4194,E1 25.1168,E2 492.8665} C_DIS
LIN {X 97.6093,Y -86.8553,Z 147,A -44.5542,B 24.9619,C -1.4254,E1 25.1205,E2 490.9355} C_DIS
LIN {X 100.3645,Y -83.6563,Z 147,A -42.8139,B 24.9619,C -1.4243,E1 25.1236,E2 489.2058} C_DIS
LIN {X 102.5654,Y -80.9423,Z 147,A -41.1742,B 24.9615,C -1.4343,E1 25.1265,E2 487.5501} C_DIS
LIN {X 105.1194,Y -77.5967,Z 147,A -39.4565,B 24.9615,C -1.4325,E1 25.1293,E2 485.845} C_DIS
LIN {X 107.4714,Y -74.3053,Z 147,A -37.6388,B 24.9612,C -1.4399,E1 25.1323,E2 484.0186} C_DIS
LIN {X 109.8153,Y -70.7956,Z 147,A -35.7722,B 24.9608,C -1.4461,E1 25.1351,E2 482.1468} C_DIS
LIN {X 112.051,Y -67.2007,Z 147,A -33.8817,B 24.9604,C -1.4534,E1 25.1379,E2 480.2487} C_DIS
LIN {X 114.247,Y -63.3946,Z 147,A -32.0093,B 24.9603,C -1.4562,E1 25.1404,E2 478.3794} C_DIS
LIN {X 116.2619,Y -59.6157,Z 147,A -30.4053,B 24.9608,C -1.4469,E1 25.1425,E2 476.8057} C_DIS
LIN {X 117.5379,Y -57.0636,Z 147,A -28.9118,B 24.9598,C -1.464,E1 25.1444,E2 475.28} C_DIS
LIN {X 119.1573,Y -53.5943,Z 147,A -27.3278,B 24.9598,C -1.464,E1 25.1462,E2 473.7045} C_DIS
LIN {X 120.3428,Y -50.8792,Z 147,A -26.0388,B 24.9597,C -1.4675,E1 25.1476,E2 472.4144} C_DIS
LIN {X 121.5681,Y -47.8778,Z 147,A -24.5732,B 24.9593,C -1.4744,E1 25.1492,E2 470.9406} C_DIS
LIN {X 122.7663,Y -44.7145,Z 147,A -23.1317,B 24.9591,C -1.4768,E1 25.1506,E2 469.5015} C_DIS
LIN {X 123.9016,Y -41.4633,Z 147,A -21.7742,B 24.9593,C -1.4733,E1 25.1518,E2 468.1599} C_DIS
LIN {X 124.702,Y -38.9977,Z 147,A -20.5275,B 24.9588,C -1.4829,E1 25.1528,E2 466.8976} C_DIS
LIN {X 125.6141,Y -35.9515,Z 147,A -19.1445,B 24.9586,C -1.4868,E1 25.1539,E2 465.5133} C_DIS
Enddeposition()
END
